LIN {X 0,Y 530.931,Z 527.98,A -85,B 0,C 180,E1 -4418.949,E2 -4418.949} C_VEL
LIN {X 0,Y 531.115,Z 519.525,A -85,B 0,C 180,E1 -4419.907,E2 -4419.907} C_VEL
LIN {X 0,Y 531.409,Z 509.073,A -85,B 0,C 180,E1 -4420.864,E2 -4420.864} C_VEL
LIN {X 0,Y 531.637,Z 497.317,A -85,B 0,C 180,E1 -4421.727,E2 -4421.727} C_VEL
LIN {X 0,Y 531.908,Z 485.378,A -85,B 0,C 180,E1 -4422.4,E2 -4422.4} C_VEL
LIN {X 0,Y 532.176,Z 472.952,A -85,B 0,C 180,E1 -4422.927,E2 -4422.927} C_VEL
LIN {X 0,Y 532.305,Z 460.13,A -85,B 0,C 180,E1 -4423.312,E2 -4423.312} C_VEL
LIN {X 0,Y 530.817,Z 450.091,A -85,B 0,C 180,E1 -4423.545,E2 -4423.545} C_VEL
LIN {X 0,Y 530.994,Z 438.88,A -85,B 0,C 180,E1 -4426.139,E2 -4426.139} C_VEL
LIN {X 0,Y 531.195,Z 426.982,A -85,B 0,C 180,E1 -4428.915,E2 -4428.915} C_VEL
LIN {X 0,Y 531.44,Z 413.99,A -85,B 0,C 180,E1 -4431.982,E2 -4431.982} C_VEL
LIN {X 0,Y 531.748,Z 401.681,A -85,B 0,C 180,E1 -4435.021,E2 -4435.021} C_VEL
LIN {X 0,Y 532.105,Z 389.883,A -85,B 0,C 180,E1 -4438.021,E2 -4438.021} C_VEL
LIN {X 0,Y 532.29,Z 381.917,A -85,B 0,C 180,E1 -4440.115,E2 -4440.115} C_VEL
LIN {X 0,Y 531.009,Z 374.342,A -85,B 0,C 180,E1 -4442.295,E2 -4442.295} C_VEL
LIN {X 0,Y 530.976,Z 374.348,A -85,B 0,C 180,E1 -4444.851,E2 -4444.851} C_VEL
LIN {X 0,Y 530.97,Z 374.344,A -85,B 0,C 180,E1 -4447.508,E2 -4447.508} C_VEL
LIN {X 0,Y 530.953,Z 374.346,A -85,B 0,C 180,E1 -4450.437,E2 -4450.437} C_VEL
LIN {X 0,Y 530.924,Z 374.354,A -85,B 0,C 180,E1 -4453.5,E2 -4453.5} C_VEL
LIN {X 0,Y 530.968,Z 374.344,A -85,B 0,C 180,E1 -4455.624,E2 -4455.624} C_VEL
LIN {X 0,Y 530.968,Z 374.345,A -85,B 0,C 180,E1 -4458.562,E2 -4458.562} C_VEL
LIN {X 0,Y 530.96,Z 374.342,A -85,B 0,C 180,E1 -4461.529,E2 -4461.529} C_VEL
LIN {X 0,Y 530.959,Z 374.35,A -85,B 0,C 180,E1 -4464.38,E2 -4464.38} C_VEL
LIN {X 0,Y 530.972,Z 374.342,A -85,B 0,C 180,E1 -4467.133,E2 -4467.133} C_VEL
LIN {X 0,Y 530.956,Z 374.35,A -85,B 0,C 180,E1 -4469.802,E2 -4469.802} C_VEL
LIN {X 0,Y 530.96,Z 374.344,A -85,B 0,C 180,E1 -4472.48,E2 -4472.48} C_VEL
LIN {X 0,Y 530.949,Z 374.345,A -85,B 0,C 180,E1 -4475.774,E2 -4475.774} C_VEL
LIN {X 0,Y 531.002,Z 374.341,A -85,B 0,C 180,E1 -4479.062,E2 -4479.062} C_VEL
LIN {X 0,Y 530.991,Z 374.34,A -85,B 0,C 180,E1 -4481.479,E2 -4481.479} C_VEL
LIN {X 0,Y 530.999,Z 374.34,A -85,B 0,C 180,E1 -4484.65,E2 -4484.65} C_VEL
LIN {X 0,Y 531.029,Z 374.341,A -85,B 0,C 180,E1 -4487.775,E2 -4487.775} C_VEL
LIN {X 0,Y 530.967,Z 374.344,A -85,B 0,C 180,E1 -4490.091,E2 -4490.091} C_VEL
LIN {X 0,Y 531.015,Z 374.343,A -85,B 0,C 180,E1 -4493.159,E2 -4493.159} C_VEL
LIN {X 0,Y 531.104,Z 374.333,A -85,B 0,C 180,E1 -4494.685,E2 -4494.685} C_VEL
LIN {X 0,Y 530.727,Z 374.457,A -85,B 0,C 180,E1 -4497.058,E2 -4497.058} C_VEL
LIN {X 0,Y 530.921,Z 382.02,A -85,B 0,C 180,E1 -4500,E2 -4500} C_VEL
LIN {X 0,Y 530.728,Z 387.746,A -85,B 0,C 180,E1 -4502.277,E2 -4502.277} C_VEL
LIN {X 0,Y 530.796,Z 395.171,A -85,B 0,C 180,E1 -4505.318,E2 -4505.318} C_VEL
LIN {X 0,Y 530.761,Z 402.54,A -85,B 0,C 180,E1 -4508.375,E2 -4508.375} C_VEL
LIN {X 0,Y 530.722,Z 409.772,A -85,B 0,C 180,E1 -4511.496,E2 -4511.496} C_VEL
LIN {X 0,Y 530.607,Z 417.392,A -85,B 0,C 180,E1 -4514.781,E2 -4514.781} C_VEL
LIN {X 0,Y 530.507,Z 423.618,A -85,B 0,C 180,E1 -4517.537,E2 -4517.537} C_VEL
LIN {X 0,Y 532.297,Z 434.899,A -85,B 0,C 180,E1 -4517.857,E2 -4517.857} C_VEL
LIN {X 0,Y 532.11,Z 445.401,A -85,B 0,C 180,E1 -4518.206,E2 -4518.206} C_VEL
LIN {X 0,Y 531.843,Z 456.316,A -85,B 0,C 180,E1 -4518.69,E2 -4518.69} C_VEL
LIN {X 0,Y 531.666,Z 466.992,A -85,B 0,C 180,E1 -4519.297,E2 -4519.297} C_VEL
LIN {X 0,Y 531.396,Z 479.241,A -85,B 0,C 180,E1 -4520.194,E2 -4520.194} C_VEL
LIN {X 0,Y 531.179,Z 487.4,A -85,B 0,C 180,E1 -4520.93,E2 -4520.93} C_VEL
LIN {X 0,Y 531.018,Z 495.07,A -85,B 0,C 180,E1 -4521.751,E2 -4521.751} C_VEL
LIN {X 0,Y 530.803,Z 503.072,A -85,B 0,C 180,E1 -4522.785,E2 -4522.785} C_VEL
LIN {X 0,Y 530.72,Z 508.892,A -85,B 0,C 180,E1 -4523.683,E2 -4523.683} C_VEL
LIN {X 0,Y 530.572,Z 514.196,A -85,B 0,C 180,E1 -4524.661,E2 -4524.661} C_VEL
LIN {X 0,Y 530.495,Z 519.722,A -85,B 0,C 180,E1 -4525.924,E2 -4525.924} C_VEL
LIN {X 0,Y 530.446,Z 524.375,A -85,B 0,C 180,E1 -4527.414,E2 -4527.414} C_VEL
LIN {X 0,Y 530.399,Z 527.522,A -85,B 0,C 180,E1 -4529.01,E2 -4529.01} C_VEL
LIN {X 0,Y 530.384,Z 528.904,A -85,B 0,C 180,E1 -4530.536,E2 -4530.536} C_VEL
LIN {X 0,Y 530.378,Z 528.658,A -85,B 0,C 180,E1 -4532.008,E2 -4532.008} C_VEL
LIN {X 0,Y 530.368,Z 527.083,A -85,B 0,C 180,E1 -4533.402,E2 -4533.402} C_VEL
LIN {X 0,Y 530.425,Z 524.169,A -85,B 0,C 180,E1 -4534.765,E2 -4534.765} C_VEL
LIN {X 0,Y 530.503,Z 519.993,A -85,B 0,C 180,E1 -4536.087,E2 -4536.087} C_VEL
LIN {X 0,Y 530.589,Z 514.554,A -85,B 0,C 180,E1 -4537.368,E2 -4537.368} C_VEL
LIN {X 0,Y 530.61,Z 512.566,A -85,B 0,C 180,E1 -4537.759,E2 -4537.759} C_VEL
LIN {X 0,Y 529.975,Z 509.631,A -85,B 0,C 180,E1 -4538.31,E2 -4538.31} C_VEL
LIN {X 0,Y 527.214,Z 504.519,A -85,B 0,C 180,E1 -4539.183,E2 -4539.183} C_VEL
LIN {X 0,Y 524.518,Z 498.801,A -85,B 0,C 180,E1 -4540.017,E2 -4540.017} C_VEL
LIN {X 0,Y 523.985,Z 494.917,A -85,B 0,C 180,E1 -4540.501,E2 -4540.501} C_VEL
LIN {X 0,Y 524.222,Z 485.978,A -85,B 0,C 180,E1 -4541.449,E2 -4541.449} C_VEL
LIN {X 0,Y 524.451,Z 476.161,A -85,B 0,C 180,E1 -4542.302,E2 -4542.302} C_VEL
LIN {X 0,Y 524.7,Z 464.968,A -85,B 0,C 180,E1 -4543.087,E2 -4543.087} C_VEL
LIN {X 0,Y 524.982,Z 453.047,A -85,B 0,C 180,E1 -4543.735,E2 -4543.735} C_VEL
LIN {X 0,Y 525.289,Z 439.587,A -85,B 0,C 180,E1 -4544.272,E2 -4544.272} C_VEL
LIN {X 0,Y 525.146,Z 433.464,A -85,B 0,C 180,E1 -4544.464,E2 -4544.464} C_VEL
LIN {X 0,Y 523.424,Z 423.693,A -85,B 0,C 180,E1 -4544.738,E2 -4544.738} C_VEL
LIN {X 0,Y 523.487,Z 417.312,A -85,B 0,C 180,E1 -4547.594,E2 -4547.594} C_VEL
LIN {X 0,Y 523.565,Z 410.89,A -85,B 0,C 180,E1 -4550.403,E2 -4550.403} C_VEL
LIN {X 0,Y 523.64,Z 403.479,A -85,B 0,C 180,E1 -4553.637,E2 -4553.637} C_VEL
LIN {X 0,Y 523.705,Z 396.674,A -85,B 0,C 180,E1 -4556.617,E2 -4556.617} C_VEL
LIN {X 0,Y 523.769,Z 390.415,A -85,B 0,C 180,E1 -4559.342,E2 -4559.342} C_VEL
LIN {X 0,Y 523.781,Z 383.555,A -85,B 0,C 180,E1 -4562.322,E2 -4562.322} C_VEL
LIN {X 0,Y 523.889,Z 376.361,A -85,B 0,C 180,E1 -4565.425,E2 -4565.425} C_VEL
LIN {X 0,Y 523.971,Z 375.22,A -85,B 0,C 180,E1 -4565.962,E2 -4565.962} C_VEL
LIN {X 0,Y 523.948,Z 375.223,A -85,B 0,C 180,E1 -4568.765,E2 -4568.765} C_VEL
LIN {X 0,Y 523.937,Z 375.22,A -85,B 0,C 180,E1 -4571.219,E2 -4571.219} C_VEL
LIN {X 0,Y 523.93,Z 375.226,A -85,B 0,C 180,E1 -4573.637,E2 -4573.637} C_VEL
LIN {X 0,Y 523.941,Z 375.219,A -85,B 0,C 180,E1 -4576.027,E2 -4576.027} C_VEL
LIN {X 0,Y 524.014,Z 375.215,A -85,B 0,C 180,E1 -4578.393,E2 -4578.393} C_VEL
LIN {X 0,Y 524.001,Z 375.217,A -85,B 0,C 180,E1 -4581.514,E2 -4581.514} C_VEL
LIN {X 0,Y 524.073,Z 375.209,A -85,B 0,C 180,E1 -4584.612,E2 -4584.612} C_VEL
LIN {X 0,Y 524.106,Z 375.204,A -85,B 0,C 180,E1 -4587.693,E2 -4587.693} C_VEL
LIN {X 0,Y 524.117,Z 375.253,A -85,B 0,C 180,E1 -4590.286,E2 -4590.286} C_VEL
LIN {X 0,Y 524.079,Z 379.167,A -85,B 0,C 180,E1 -4592.304,E2 -4592.304} C_VEL
LIN {X 0,Y 523.878,Z 385.251,A -85,B 0,C 180,E1 -4595.387,E2 -4595.387} C_VEL
LIN {X 0,Y 523.809,Z 389.903,A -85,B 0,C 180,E1 -4597.709,E2 -4597.709} C_VEL
LIN {X 0,Y 523.734,Z 396.172,A -85,B 0,C 180,E1 -4600.826,E2 -4600.826} C_VEL
LIN {X 0,Y 523.615,Z 402.623,A -85,B 0,C 180,E1 -4603.979,E2 -4603.979} C_VEL
LIN {X 0,Y 523.496,Z 409.248,A -85,B 0,C 180,E1 -4607.176,E2 -4607.176} C_VEL
LIN {X 0,Y 523.382,Z 416.011,A -85,B 0,C 180,E1 -4610.432,E2 -4610.432} C_VEL
LIN {X 0,Y 523.417,Z 419.782,A -85,B 0,C 180,E1 -4612.22,E2 -4612.22} C_VEL
LIN {X 0,Y 524.68,Z 430.393,A -85,B 0,C 180,E1 -4612.57,E2 -4612.57} C_VEL
LIN {X 0,Y 524.396,Z 441.937,A -85,B 0,C 180,E1 -4613.077,E2 -4613.077} C_VEL
LIN {X 0,Y 524.2,Z 450.946,A -85,B 0,C 180,E1 -4613.609,E2 -4613.609} C_VEL
LIN {X 0,Y 524.051,Z 459.242,A -85,B 0,C 180,E1 -4614.226,E2 -4614.226} C_VEL
LIN {X 0,Y 523.927,Z 466.514,A -85,B 0,C 180,E1 -4614.887,E2 -4614.887} C_VEL
LIN {X 0,Y 523.77,Z 472.963,A -85,B 0,C 180,E1 -4615.591,E2 -4615.591} C_VEL
LIN {X 0,Y 523.648,Z 479.751,A -85,B 0,C 180,E1 -4616.501,E2 -4616.501} C_VEL
LIN {X 0,Y 523.529,Z 485.076,A -85,B 0,C 180,E1 -4617.38,E2 -4617.38} C_VEL
LIN {X 0,Y 523.502,Z 488.386,A -85,B 0,C 180,E1 -4618.023,E2 -4618.023} C_VEL
LIN {X 0,Y 523.448,Z 493.123,A -85,B 0,C 180,E1 -4619.225,E2 -4619.225} C_VEL
LIN {X 0,Y 523.384,Z 496.023,A -85,B 0,C 180,E1 -4620.232,E2 -4620.232} C_VEL
LIN {X 0,Y 523.311,Z 497.153,A -85,B 0,C 180,E1 -4620.739,E2 -4620.739} C_VEL
LIN {X 0,Y 523.263,Z 499.086,A -85,B 0,C 180,E1 -4622.204,E2 -4622.204} C_VEL
LIN {X 0,Y 523.294,Z 499.2,A -85,B 0,C 180,E1 -4623.626,E2 -4623.626} C_VEL
LIN {X 0,Y 523.291,Z 498.686,A -85,B 0,C 180,E1 -4624.335,E2 -4624.335} C_VEL
LIN {X 0,Y 523.311,Z 497.339,A -85,B 0,C 180,E1 -4625.271,E2 -4625.271} C_VEL
LIN {X 0,Y 523.396,Z 494.851,A -85,B 0,C 180,E1 -4626.326,E2 -4626.326} C_VEL
LIN {X 0,Y 523.438,Z 492.137,A -85,B 0,C 180,E1 -4627.168,E2 -4627.168} C_VEL
LIN {X 0,Y 523.506,Z 488.098,A -85,B 0,C 180,E1 -4628.134,E2 -4628.134} C_VEL
LIN {X 0,Y 523.605,Z 482.896,A -85,B 0,C 180,E1 -4629.109,E2 -4629.109} C_VEL
LIN {X 0,Y 523.755,Z 476.136,A -85,B 0,C 180,E1 -4630.106,E2 -4630.106} C_VEL
LIN {X 0,Y 523.862,Z 468.849,A -85,B 0,C 180,E1 -4630.969,E2 -4630.969} C_VEL
LIN {X 0,Y 524.025,Z 461.627,A -85,B 0,C 180,E1 -4631.668,E2 -4631.668} C_VEL
LIN {X 0,Y 524.242,Z 453.662,A -85,B 0,C 180,E1 -4632.298,E2 -4632.298} C_VEL
LIN {X 0,Y 524.421,Z 445.007,A -85,B 0,C 180,E1 -4632.849,E2 -4632.849} C_VEL
LIN {X 0,Y 524.56,Z 436.043,A -85,B 0,C 180,E1 -4633.296,E2 -4633.296} C_VEL
LIN {X 0,Y 524.48,Z 427.33,A -85,B 0,C 180,E1 -4633.631,E2 -4633.631} C_VEL
LIN {X 0,Y 523.402,Z 419.767,A -85,B 0,C 180,E1 -4633.89,E2 -4633.89} C_VEL
LIN {X 0,Y 523.452,Z 413.7,A -85,B 0,C 180,E1 -4636.785,E2 -4636.785} C_VEL
LIN {X 0,Y 523.488,Z 408.426,A -85,B 0,C 180,E1 -4639.374,E2 -4639.374} C_VEL
LIN {X 0,Y 523.587,Z 402.331,A -85,B 0,C 180,E1 -4642.363,E2 -4642.363} C_VEL
LIN {X 0,Y 523.658,Z 397.039,A -85,B 0,C 180,E1 -4644.948,E2 -4644.948} C_VEL
LIN {X 0,Y 523.73,Z 391.464,A -85,B 0,C 180,E1 -4647.71,E2 -4647.71} C_VEL
LIN {X 0,Y 523.83,Z 385.498,A -85,B 0,C 180,E1 -4650.695,E2 -4650.695} C_VEL
LIN {X 0,Y 523.929,Z 381.209,A -85,B 0,C 180,E1 -4652.866,E2 -4652.866} C_VEL
LIN {X 0,Y 524.023,Z 375.454,A -85,B 0,C 180,E1 -4655.774,E2 -4655.774} C_VEL
LIN {X 0,Y 523.965,Z 375.222,A -85,B 0,C 180,E1 -4656.272,E2 -4656.272} C_VEL
LIN {X 0,Y 523.936,Z 375.223,A -85,B 0,C 180,E1 -4658.767,E2 -4658.767} C_VEL
LIN {X 0,Y 523.933,Z 375.224,A -85,B 0,C 180,E1 -4661.22,E2 -4661.22} C_VEL
LIN {X 0,Y 523.918,Z 375.226,A -85,B 0,C 180,E1 -4663.639,E2 -4663.639} C_VEL
LIN {X 0,Y 523.929,Z 375.226,A -85,B 0,C 180,E1 -4666.028,E2 -4666.028} C_VEL
LIN {X 0,Y 523.995,Z 375.216,A -85,B 0,C 180,E1 -4668.394,E2 -4668.394} C_VEL
LIN {X 0,Y 523.986,Z 375.217,A -85,B 0,C 180,E1 -4671.516,E2 -4671.516} C_VEL
LIN {X 0,Y 524.083,Z 375.203,A -85,B 0,C 180,E1 -4674.614,E2 -4674.614} C_VEL
LIN {X 0,Y 524.095,Z 375.203,A -85,B 0,C 180,E1 -4677.695,E2 -4677.695} C_VEL
LIN {X 0,Y 524.106,Z 375.202,A -85,B 0,C 180,E1 -4680.769,E2 -4680.769} C_VEL
LIN {X 0,Y 524.056,Z 375.208,A -85,B 0,C 180,E1 -4683.075,E2 -4683.075} C_VEL
LIN {X 0,Y 524.032,Z 375.21,A -85,B 0,C 180,E1 -4686.159,E2 -4686.159} C_VEL
LIN {X 0,Y 523.988,Z 375.214,A -85,B 0,C 180,E1 -4689.262,E2 -4689.262} C_VEL
LIN {X 0,Y 524.019,Z 375.211,A -85,B 0,C 180,E1 -4691.763,E2 -4691.763} C_VEL
LIN {X 0,Y 523.97,Z 375.218,A -85,B 0,C 180,E1 -4695.054,E2 -4695.054} C_VEL
LIN {X 0,Y 523.948,Z 375.223,A -85,B 0,C 180,E1 -4697.97,E2 -4697.97} C_VEL
LIN {X 0,Y 523.951,Z 375.221,A -85,B 0,C 180,E1 -4700.411,E2 -4700.411} C_VEL
LIN {X 0,Y 523.929,Z 375.223,A -85,B 0,C 180,E1 -4702.893,E2 -4702.893} C_VEL
LIN {X 0,Y 523.965,Z 375.221,A -85,B 0,C 180,E1 -4706.022,E2 -4706.022} C_VEL
LIN {X 0,Y 523.931,Z 375.223,A -85,B 0,C 180,E1 -4708.875,E2 -4708.875} C_VEL
LIN {X 0,Y 523.913,Z 375.225,A -85,B 0,C 180,E1 -4711.545,E2 -4711.545} C_VEL
LIN {X 0,Y 523.928,Z 375.224,A -85,B 0,C 180,E1 -4714.291,E2 -4714.291} C_VEL
LIN {X 0,Y 523.894,Z 375.227,A -85,B 0,C 180,E1 -4717.134,E2 -4717.134} C_VEL
LIN {X 0,Y 523.952,Z 375.22,A -85,B 0,C 180,E1 -4720.136,E2 -4720.136} C_VEL
LIN {X 0,Y 523.912,Z 375.227,A -85,B 0,C 180,E1 -4723.168,E2 -4723.168} C_VEL
LIN {X 0,Y 523.927,Z 375.223,A -85,B 0,C 180,E1 -4725.774,E2 -4725.774} C_VEL
LIN {X 0,Y 523.949,Z 375.223,A -85,B 0,C 180,E1 -4728.912,E2 -4728.912} C_VEL
LIN {X 0,Y 523.906,Z 375.226,A -85,B 0,C 180,E1 -4731.901,E2 -4731.901} C_VEL
LIN {X 0,Y 523.93,Z 375.224,A -85,B 0,C 180,E1 -4734.911,E2 -4734.911} C_VEL
LIN {X 0,Y 523.975,Z 375.332,A -85,B 0,C 180,E1 -4737.442,E2 -4737.442} C_VEL
LIN {X 0,Y 525.212,Z 382.036,A -85,B 0,C 180,E1 -4739.44,E2 -4739.44} C_VEL
LIN {X 0,Y 525.262,Z 386.946,A -85,B 0,C 180,E1 -4740.805,E2 -4740.805} C_VEL
LIN {X 0,Y 524.915,Z 396.536,A -85,B 0,C 180,E1 -4743.353,E2 -4743.353} C_VEL
LIN {X 0,Y 524.574,Z 408.028,A -85,B 0,C 180,E1 -4746.304,E2 -4746.304} C_VEL
LIN {X 0,Y 524.243,Z 419.584,A -85,B 0,C 180,E1 -4749.193,E2 -4749.193} C_VEL
LIN {X 0,Y 524.036,Z 432.384,A -85,B 0,C 180,E1 -4752.214,E2 -4752.214} C_VEL
LIN {X 0,Y 523.855,Z 445.336,A -85,B 0,C 180,E1 -4755.234,E2 -4755.234} C_VEL
LIN {X 0,Y 523.765,Z 449.924,A -85,B 0,C 180,E1 -4756.298,E2 -4756.298} C_VEL
LIN {X 0,Y 525.384,Z 461.083,A -85,B 0,C 180,E1 -4756.562,E2 -4756.562} C_VEL
LIN {X 0,Y 525.185,Z 473.533,A -85,B 0,C 180,E1 -4756.951,E2 -4756.951} C_VEL
LIN {X 0,Y 524.916,Z 484.759,A -85,B 0,C 180,E1 -4757.436,E2 -4757.436} C_VEL
LIN {X 0,Y 524.636,Z 496.338,A -85,B 0,C 180,E1 -4758.087,E2 -4758.087} C_VEL
LIN {X 0,Y 524.442,Z 507.516,A -85,B 0,C 180,E1 -4758.895,E2 -4758.895} C_VEL
LIN {X 0,Y 524.157,Z 517.303,A -85,B 0,C 180,E1 -4759.769,E2 -4759.769} C_VEL
LIN {X 0,Y 523.928,Z 526.218,A -85,B 0,C 180,E1 -4760.739,E2 -4760.739} C_VEL
LIN {X 0,Y 523.722,Z 534.907,A -85,B 0,C 180,E1 -4761.902,E2 -4761.902} C_VEL
LIN {X 0,Y 523.573,Z 541.849,A -85,B 0,C 180,E1 -4763.063,E2 -4763.063} C_VEL
LIN {X 0,Y 523.543,Z 547.372,A -85,B 0,C 180,E1 -4764.224,E2 -4764.224} C_VEL
LIN {X 0,Y 523.36,Z 551.682,A -85,B 0,C 180,E1 -4765.38,E2 -4765.38} C_VEL
LIN {X 0,Y 523.443,Z 553.965,A -85,B 0,C 180,E1 -4766.153,E2 -4766.153} C_VEL
LIN {X 0,Y 523.367,Z 555.814,A -85,B 0,C 180,E1 -4766.923,E2 -4766.923} C_VEL
LIN {X 0,Y 523.335,Z 557.198,A -85,B 0,C 180,E1 -4767.693,E2 -4767.693} C_VEL
LIN {X 0,Y 523.25,Z 558.787,A -85,B 0,C 180,E1 -4769.232,E2 -4769.232} C_VEL
LIN {X 0,Y 523.246,Z 559,A -85,B 0,C 180,E1 -4770.002,E2 -4770.002} C_VEL
LIN {X 0,Y 523.275,Z 558.18,A -85,B 0,C 180,E1 -4771.541,E2 -4771.541} C_VEL
LIN {X 0,Y 523.335,Z 557.19,A -85,B 0,C 180,E1 -4772.311,E2 -4772.311} C_VEL
LIN {X 0,Y 523.368,Z 555.803,A -85,B 0,C 180,E1 -4773.081,E2 -4773.081} C_VEL
LIN {X 0,Y 523.442,Z 552.889,A -85,B 0,C 180,E1 -4774.237,E2 -4774.237} C_VEL
LIN {X 0,Y 523.465,Z 548.944,A -85,B 0,C 180,E1 -4775.394,E2 -4775.394} C_VEL
LIN {X 0,Y 523.525,Z 543.706,A -85,B 0,C 180,E1 -4776.582,E2 -4776.582} C_VEL
LIN {X 0,Y 523.667,Z 537.376,A -85,B 0,C 180,E1 -4777.714,E2 -4777.714} C_VEL
LIN {X 0,Y 523.846,Z 529.297,A -85,B 0,C 180,E1 -4778.877,E2 -4778.877} C_VEL
LIN {X 0,Y 524.057,Z 521.061,A -85,B 0,C 180,E1 -4779.847,E2 -4779.847} C_VEL
LIN {X 0,Y 524.316,Z 511.016,A -85,B 0,C 180,E1 -4780.818,E2 -4780.818} C_VEL
LIN {X 0,Y 524.632,Z 499.723,A -85,B 0,C 180,E1 -4781.686,E2 -4781.686} C_VEL
LIN {X 0,Y 524.831,Z 488.494,A -85,B 0,C 180,E1 -4782.373,E2 -4782.373} C_VEL
LIN {X 0,Y 525.135,Z 476.104,A -85,B 0,C 180,E1 -4782.955,E2 -4782.955} C_VEL
LIN {X 0,Y 525.363,Z 462.889,A -85,B 0,C 180,E1 -4783.392,E2 -4783.392} C_VEL
LIN {X 0,Y 524.977,Z 457.876,A -85,B 0,C 180,E1 -4783.526,E2 -4783.526} C_VEL
LIN {X 0,Y 523.756,Z 449.781,A -85,B 0,C 180,E1 -4783.731,E2 -4783.731} C_VEL
LIN {X 0,Y 523.945,Z 438.566,A -85,B 0,C 180,E1 -4786.362,E2 -4786.362} C_VEL
LIN {X 0,Y 524.147,Z 426.663,A -85,B 0,C 180,E1 -4789.179,E2 -4789.179} C_VEL
LIN {X 0,Y 524.441,Z 414.908,A -85,B 0,C 180,E1 -4792.04,E2 -4792.04} C_VEL
LIN {X 0,Y 524.766,Z 403.24,A -85,B 0,C 180,E1 -4794.954,E2 -4794.954} C_VEL
LIN {X 0,Y 525.183,Z 390.057,A -85,B 0,C 180,E1 -4798.364,E2 -4798.364} C_VEL
LIN {X 0,Y 525.367,Z 383.542,A -85,B 0,C 180,E1 -4800.11,E2 -4800.11} C_VEL
LIN {X 0,Y 523.958,Z 375.222,A -85,B 0,C 180,E1 -4802.534,E2 -4802.534} C_VEL
LIN {X 0,Y 523.925,Z 375.223,A -85,B 0,C 180,E1 -4805.227,E2 -4805.227} C_VEL
LIN {X 0,Y 523.919,Z 375.227,A -85,B 0,C 180,E1 -4808.103,E2 -4808.103} C_VEL
LIN {X 0,Y 523.92,Z 375.222,A -85,B 0,C 180,E1 -4811.305,E2 -4811.305} C_VEL
LIN {X 0,Y 523.936,Z 375.219,A -85,B 0,C 180,E1 -4814.689,E2 -4814.689} C_VEL
LIN {X 0,Y 523.913,Z 375.221,A -85,B 0,C 180,E1 -4817.877,E2 -4817.877} C_VEL
LIN {X 0,Y 523.921,Z 375.222,A -85,B 0,C 180,E1 -4821.081,E2 -4821.081} C_VEL
LIN {X 0,Y 523.906,Z 375.223,A -85,B 0,C 180,E1 -4823.825,E2 -4823.825} C_VEL
LIN {X 0,Y 523.918,Z 375.222,A -85,B 0,C 180,E1 -4826.634,E2 -4826.634} C_VEL
LIN {X 0,Y 523.949,Z 375.219,A -85,B 0,C 180,E1 -4829.355,E2 -4829.355} C_VEL
LIN {X 0,Y 523.917,Z 375.221,A -85,B 0,C 180,E1 -4832.295,E2 -4832.295} C_VEL
LIN {X 0,Y 523.897,Z 375.226,A -85,B 0,C 180,E1 -4835.426,E2 -4835.426} C_VEL
LIN {X 0,Y 523.942,Z 375.218,A -85,B 0,C 180,E1 -4837.939,E2 -4837.939} C_VEL
LIN {X 0,Y 523.978,Z 375.22,A -85,B 0,C 180,E1 -4840.408,E2 -4840.408} C_VEL
LIN {X 0,Y 523.971,Z 375.216,A -85,B 0,C 180,E1 -4842.837,E2 -4842.837} C_VEL
LIN {X 0,Y 523.981,Z 375.215,A -85,B 0,C 180,E1 -4845.236,E2 -4845.236} C_VEL
LIN {X 0,Y 524.017,Z 375.209,A -85,B 0,C 180,E1 -4848.394,E2 -4848.394} C_VEL
LIN {X 0,Y 523.948,Z 375.222,A -85,B 0,C 180,E1 -4851.515,E2 -4851.515} C_VEL
LIN {X 0,Y 524.048,Z 375.211,A -85,B 0,C 180,E1 -4854.613,E2 -4854.613} C_VEL
LIN {X 0,Y 523.669,Z 375.428,A -85,B 0,C 180,E1 -4857.115,E2 -4857.115} C_VEL
LIN {X 0,Y 523.879,Z 382.806,A -85,B 0,C 180,E1 -4860,E2 -4860} C_VEL
LIN {X 0,Y 523.662,Z 388.565,A -85,B 0,C 180,E1 -4862.307,E2 -4862.307} C_VEL
LIN {X 0,Y 523.744,Z 394.199,A -85,B 0,C 180,E1 -4864.618,E2 -4864.618} C_VEL
LIN {X 0,Y 523.679,Z 401.576,A -85,B 0,C 180,E1 -4867.712,E2 -4867.712} C_VEL
LIN {X 0,Y 523.619,Z 407.094,A -85,B 0,C 180,E1 -4870.048,E2 -4870.048} C_VEL
LIN {X 0,Y 523.572,Z 412.511,A -85,B 0,C 180,E1 -4872.402,E2 -4872.402} C_VEL
LIN {X 0,Y 523.522,Z 418.186,A -85,B 0,C 180,E1 -4874.858,E2 -4874.858} C_VEL
LIN {X 0,Y 523.445,Z 423.749,A -85,B 0,C 180,E1 -4877.352,E2 -4877.352} C_VEL
LIN {X 0,Y 525.37,Z 435.711,A -85,B 0,C 180,E1 -4877.699,E2 -4877.699} C_VEL
LIN {X 0,Y 525.152,Z 448.719,A -85,B 0,C 180,E1 -4878.161,E2 -4878.161} C_VEL
LIN {X 0,Y 524.83,Z 460.623,A -85,B 0,C 180,E1 -4878.746,E2 -4878.746} C_VEL
LIN {X 0,Y 524.598,Z 471.88,A -85,B 0,C 180,E1 -4879.466,E2 -4879.466} C_VEL
LIN {X 0,Y 524.355,Z 481.646,A -85,B 0,C 180,E1 -4880.244,E2 -4880.244} C_VEL
LIN {X 0,Y 524.113,Z 489.742,A -85,B 0,C 180,E1 -4881.02,E2 -4881.02} C_VEL
LIN {X 0,Y 523.901,Z 497.087,A -85,B 0,C 180,E1 -4881.855,E2 -4881.855} C_VEL
LIN {X 0,Y 523.736,Z 504.746,A -85,B 0,C 180,E1 -4882.901,E2 -4882.901} C_VEL
LIN {X 0,Y 523.592,Z 510.906,A -85,B 0,C 180,E1 -4883.922,E2 -4883.922} C_VEL
LIN {X 0,Y 523.44,Z 516.33,A -85,B 0,C 180,E1 -4885.02,E2 -4885.02} C_VEL
LIN {X 0,Y 523.409,Z 521.329,A -85,B 0,C 180,E1 -4886.302,E2 -4886.302} C_VEL
LIN {X 0,Y 523.335,Z 524.976,A -85,B 0,C 180,E1 -4887.583,E2 -4887.583} C_VEL
LIN {X 0,Y 523.305,Z 527.778,A -85,B 0,C 180,E1 -4889.196,E2 -4889.196} C_VEL
LIN {X 0,Y 523.315,Z 528.473,A -85,B 0,C 180,E1 -4889.795,E2 -4889.795} C_VEL
LIN {X 0,Y 523.281,Z 528.947,A -85,B 0,C 180,E1 -4890.732,E2 -4890.732} C_VEL
LIN {X 0,Y 523.272,Z 528.55,A -85,B 0,C 180,E1 -4892.204,E2 -4892.204} C_VEL
LIN {X 0,Y 523.292,Z 526.766,A -85,B 0,C 180,E1 -4893.624,E2 -4893.624} C_VEL
LIN {X 0,Y 523.329,Z 523.715,A -85,B 0,C 180,E1 -4894.995,E2 -4894.995} C_VEL
LIN {X 0,Y 523.426,Z 519.412,A -85,B 0,C 180,E1 -4896.329,E2 -4896.329} C_VEL
LIN {X 0,Y 523.532,Z 513.794,A -85,B 0,C 180,E1 -4897.624,E2 -4897.624} C_VEL
LIN {X 0,Y 523.638,Z 506.783,A -85,B 0,C 180,E1 -4898.881,E2 -4898.881} C_VEL
LIN {X 0,Y 523.864,Z 498.325,A -85,B 0,C 180,E1 -4900.087,E2 -4900.087} C_VEL
LIN {X 0,Y 523.985,Z 494.917,A -85,B 0,C 180,E1 -4900.501,E2 -4900.501} C_VEL
LIN {X 0,Y 523.445,Z 490.873,A -85,B 0,C 180,E1 -4900.968,E2 -4900.968} C_VEL
LIN {X 0,Y 520.748,Z 484.101,A -85,B 0,C 180,E1 -4901.71,E2 -4901.71} C_VEL
LIN {X 0,Y 518.081,Z 476.865,A -85,B 0,C 180,E1 -4902.398,E2 -4902.398} C_VEL
LIN {X 0,Y 517.579,Z 472.072,A -85,B 0,C 180,E1 -4902.775,E2 -4902.775} C_VEL
LIN {X 0,Y 517.872,Z 460.337,A -85,B 0,C 180,E1 -4903.531,E2 -4903.531} C_VEL
LIN {X 0,Y 518.181,Z 448.806,A -85,B 0,C 180,E1 -4904.103,E2 -4904.103} C_VEL
LIN {X 0,Y 518.424,Z 435.768,A -85,B 0,C 180,E1 -4904.573,E2 -4904.573} C_VEL
LIN {X 0,Y 516.35,Z 423.831,A -85,B 0,C 180,E1 -4904.928,E2 -4904.928} C_VEL
LIN {X 0,Y 516.415,Z 418.568,A -85,B 0,C 180,E1 -4907.298,E2 -4907.298} C_VEL
LIN {X 0,Y 516.501,Z 411.881,A -85,B 0,C 180,E1 -4910.242,E2 -4910.242} C_VEL
LIN {X 0,Y 516.558,Z 404.748,A -85,B 0,C 180,E1 -4913.39,E2 -4913.39} C_VEL
LIN {X 0,Y 516.655,Z 398.582,A -85,B 0,C 180,E1 -4916.101,E2 -4916.101} C_VEL
LIN {X 0,Y 516.71,Z 392.061,A -85,B 0,C 180,E1 -4918.969,E2 -4918.969} C_VEL
LIN {X 0,Y 516.738,Z 384.873,A -85,B 0,C 180,E1 -4922.134,E2 -4922.134} C_VEL
LIN {X 0,Y 516.805,Z 378.075,A -85,B 0,C 180,E1 -4925.065,E2 -4925.065} C_VEL
LIN {X 0,Y 516.902,Z 376.101,A -85,B 0,C 180,E1 -4925.926,E2 -4925.926} C_VEL
LIN {X 0,Y 516.888,Z 376.099,A -85,B 0,C 180,E1 -4928.461,E2 -4928.461} C_VEL
LIN {X 0,Y 516.892,Z 376.098,A -85,B 0,C 180,E1 -4930.953,E2 -4930.953} C_VEL
LIN {X 0,Y 516.905,Z 376.099,A -85,B 0,C 180,E1 -4933.409,E2 -4933.409} C_VEL
LIN {X 0,Y 516.896,Z 376.097,A -85,B 0,C 180,E1 -4935.832,E2 -4935.832} C_VEL
LIN {X 0,Y 516.95,Z 376.09,A -85,B 0,C 180,E1 -4939.026,E2 -4939.026} C_VEL
LIN {X 0,Y 516.979,Z 376.087,A -85,B 0,C 180,E1 -4942.185,E2 -4942.185} C_VEL
LIN {X 0,Y 517.02,Z 376.087,A -85,B 0,C 180,E1 -4944.538,E2 -4944.538} C_VEL
LIN {X 0,Y 517.075,Z 376.079,A -85,B 0,C 180,E1 -4947.661,E2 -4947.661} C_VEL
LIN {X 0,Y 517.089,Z 376.227,A -85,B 0,C 180,E1 -4950.29,E2 -4950.29} C_VEL
LIN {X 0,Y 517.044,Z 380.165,A -85,B 0,C 180,E1 -4952.335,E2 -4952.335} C_VEL
LIN {X 0,Y 516.834,Z 386.28,A -85,B 0,C 180,E1 -4955.46,E2 -4955.46} C_VEL
LIN {X 0,Y 516.752,Z 390.94,A -85,B 0,C 180,E1 -4957.815,E2 -4957.815} C_VEL
LIN {X 0,Y 516.672,Z 397.259,A -85,B 0,C 180,E1 -4960.976,E2 -4960.976} C_VEL
LIN {X 0,Y 516.543,Z 403.706,A -85,B 0,C 180,E1 -4964.174,E2 -4964.174} C_VEL
LIN {X 0,Y 516.416,Z 410.386,A -85,B 0,C 180,E1 -4967.419,E2 -4967.419} C_VEL
LIN {X 0,Y 516.311,Z 417.245,A -85,B 0,C 180,E1 -4970.724,E2 -4970.724} C_VEL
LIN {X 0,Y 516.354,Z 420.001,A -85,B 0,C 180,E1 -4972.049,E2 -4972.049} C_VEL
LIN {X 0,Y 517.737,Z 430.351,A -85,B 0,C 180,E1 -4972.401,E2 -4972.401} C_VEL
LIN {X 0,Y 517.492,Z 441.255,A -85,B 0,C 180,E1 -4972.874,E2 -4972.874} C_VEL
LIN {X 0,Y 517.25,Z 450.502,A -85,B 0,C 180,E1 -4973.415,E2 -4973.415} C_VEL
LIN {X 0,Y 517.076,Z 459.202,A -85,B 0,C 180,E1 -4974.061,E2 -4974.061} C_VEL
LIN {X 0,Y 516.937,Z 466.896,A -85,B 0,C 180,E1 -4974.768,E2 -4974.768} C_VEL
LIN {X 0,Y 516.727,Z 474.126,A -85,B 0,C 180,E1 -4975.581,E2 -4975.581} C_VEL
LIN {X 0,Y 516.586,Z 480.875,A -85,B 0,C 180,E1 -4976.52,E2 -4976.52} C_VEL
LIN {X 0,Y 516.42,Z 486.841,A -85,B 0,C 180,E1 -4977.559,E2 -4977.559} C_VEL
LIN {X 0,Y 516.367,Z 490.849,A -85,B 0,C 180,E1 -4978.446,E2 -4978.446} C_VEL
LIN {X 0,Y 516.362,Z 494.298,A -85,B 0,C 180,E1 -4979.416,E2 -4979.416} C_VEL
LIN {X 0,Y 516.313,Z 496.533,A -85,B 0,C 180,E1 -4980.238,E2 -4980.238} C_VEL
LIN {X 0,Y 516.197,Z 498.334,A -85,B 0,C 180,E1 -4981.153,E2 -4981.153} C_VEL
LIN {X 0,Y 516.199,Z 499.6,A -85,B 0,C 180,E1 -4982.422,E2 -4982.422} C_VEL
LIN {X 0,Y 516.189,Z 499.812,A -85,B 0,C 180,E1 -4982.995,E2 -4982.995} C_VEL
LIN {X 0,Y 516.212,Z 499.483,A -85,B 0,C 180,E1 -4983.928,E2 -4983.928} C_VEL
LIN {X 0,Y 516.239,Z 497.878,A -85,B 0,C 180,E1 -4985.232,E2 -4985.232} C_VEL
LIN {X 0,Y 516.344,Z 494.629,A -85,B 0,C 180,E1 -4986.578,E2 -4986.578} C_VEL
LIN {X 0,Y 516.385,Z 492.378,A -85,B 0,C 180,E1 -4987.272,E2 -4987.272} C_VEL
LIN {X 0,Y 516.492,Z 486.985,A -85,B 0,C 180,E1 -4988.512,E2 -4988.512} C_VEL
LIN {X 0,Y 516.602,Z 480.999,A -85,B 0,C 180,E1 -4989.561,E2 -4989.561} C_VEL
LIN {X 0,Y 516.769,Z 473.995,A -85,B 0,C 180,E1 -4990.535,E2 -4990.535} C_VEL
LIN {X 0,Y 516.942,Z 465.914,A -85,B 0,C 180,E1 -4991.433,E2 -4991.433} C_VEL
LIN {X 0,Y 517.202,Z 456.374,A -85,B 0,C 180,E1 -4992.267,E2 -4992.267} C_VEL
LIN {X 0,Y 517.44,Z 445.973,A -85,B 0,C 180,E1 -4992.963,E2 -4992.963} C_VEL
LIN {X 0,Y 517.622,Z 435.978,A -85,B 0,C 180,E1 -4993.469,E2 -4993.469} C_VEL
LIN {X 0,Y 517.541,Z 427.826,A -85,B 0,C 180,E1 -4993.787,E2 -4993.787} C_VEL
LIN {X 0,Y 516.341,Z 420.016,A -85,B 0,C 180,E1 -4994.063,E2 -4994.063} C_VEL
LIN {X 0,Y 516.387,Z 413.267,A -85,B 0,C 180,E1 -4997.298,E2 -4997.298} C_VEL
LIN {X 0,Y 516.43,Z 407.387,A -85,B 0,C 180,E1 -5000.237,E2 -5000.237} C_VEL
LIN {X 0,Y 516.538,Z 401.298,A -85,B 0,C 180,E1 -5003.226,E2 -5003.226} C_VEL
LIN {X 0,Y 516.63,Z 395.497,A -85,B 0,C 180,E1 -5006.1,E2 -5006.1} C_VEL
LIN {X 0,Y 516.719,Z 389.826,A -85,B 0,C 180,E1 -5008.962,E2 -5008.962} C_VEL
LIN {X 0,Y 516.876,Z 383.649,A -85,B 0,C 180,E1 -5012.099,E2 -5012.099} C_VEL
LIN {X 0,Y 516.971,Z 377.826,A -85,B 0,C 180,E1 -5015.075,E2 -5015.075} C_VEL
LIN {X 0,Y 516.952,Z 376.095,A -85,B 0,C 180,E1 -5016.037,E2 -5016.037} C_VEL
LIN {X 0,Y 516.893,Z 376.103,A -85,B 0,C 180,E1 -5019.298,E2 -5019.298} C_VEL
LIN {X 0,Y 516.907,Z 376.099,A -85,B 0,C 180,E1 -5022.596,E2 -5022.596} C_VEL
LIN {X 0,Y 516.926,Z 376.096,A -85,B 0,C 180,E1 -5025.03,E2 -5025.03} C_VEL
LIN {X 0,Y 516.978,Z 376.089,A -85,B 0,C 180,E1 -5028.234,E2 -5028.234} C_VEL
LIN {X 0,Y 516.95,Z 376.094,A -85,B 0,C 180,E1 -5031.4,E2 -5031.4} C_VEL
LIN {X 0,Y 517.044,Z 376.08,A -85,B 0,C 180,E1 -5034.54,E2 -5034.54} C_VEL
LIN {X 0,Y 517.066,Z 376.079,A -85,B 0,C 180,E1 -5037.663,E2 -5037.663} C_VEL
LIN {X 0,Y 517.075,Z 376.077,A -85,B 0,C 180,E1 -5040.779,E2 -5040.779} C_VEL
LIN {X 0,Y 517.023,Z 376.085,A -85,B 0,C 180,E1 -5043.117,E2 -5043.117} C_VEL
LIN {X 0,Y 516.994,Z 376.086,A -85,B 0,C 180,E1 -5046.244,E2 -5046.244} C_VEL
LIN {X 0,Y 516.943,Z 376.091,A -85,B 0,C 180,E1 -5049.39,E2 -5049.39} C_VEL
LIN {X 0,Y 516.978,Z 376.088,A -85,B 0,C 180,E1 -5051.836,E2 -5051.836} C_VEL
LIN {X 0,Y 516.923,Z 376.097,A -85,B 0,C 180,E1 -5055.149,E2 -5055.149} C_VEL
LIN {X 0,Y 516.908,Z 376.097,A -85,B 0,C 180,E1 -5058.223,E2 -5058.223} C_VEL
LIN {X 0,Y 516.895,Z 376.101,A -85,B 0,C 180,E1 -5060.702,E2 -5060.702} C_VEL
LIN {X 0,Y 516.873,Z 376.104,A -85,B 0,C 180,E1 -5063.224,E2 -5063.224} C_VEL
LIN {X 0,Y 516.924,Z 376.096,A -85,B 0,C 180,E1 -5066.198,E2 -5066.198} C_VEL
LIN {X 0,Y 516.916,Z 376.095,A -85,B 0,C 180,E1 -5069.305,E2 -5069.305} C_VEL
LIN {X 0,Y 516.882,Z 376.101,A -85,B 0,C 180,E1 -5072.546,E2 -5072.546} C_VEL
LIN {X 0,Y 516.866,Z 376.105,A -85,B 0,C 180,E1 -5075.334,E2 -5075.334} C_VEL
LIN {X 0,Y 516.865,Z 376.105,A -85,B 0,C 180,E1 -5077.945,E2 -5077.945} C_VEL
LIN {X 0,Y 516.888,Z 376.103,A -85,B 0,C 180,E1 -5080.742,E2 -5080.742} C_VEL
LIN {X 0,Y 516.869,Z 376.102,A -85,B 0,C 180,E1 -5083.905,E2 -5083.905} C_VEL
LIN {X 0,Y 516.868,Z 376.106,A -85,B 0,C 180,E1 -5086.109,E2 -5086.109} C_VEL
LIN {X 0,Y 516.892,Z 376.1,A -85,B 0,C 180,E1 -5089.263,E2 -5089.263} C_VEL
LIN {X 0,Y 516.871,Z 376.102,A -85,B 0,C 180,E1 -5092.059,E2 -5092.059} C_VEL
LIN {X 0,Y 516.887,Z 376.103,A -85,B 0,C 180,E1 -5095.179,E2 -5095.179} C_VEL
LIN {X 0,Y 516.93,Z 376.196,A -85,B 0,C 180,E1 -5097.173,E2 -5097.173} C_VEL
LIN {X 0,Y 518.29,Z 383.649,A -85,B 0,C 180,E1 -5099.439,E2 -5099.439} C_VEL
LIN {X 0,Y 518.327,Z 388.435,A -85,B 0,C 180,E1 -5100.785,E2 -5100.785} C_VEL
LIN {X 0,Y 517.87,Z 398.845,A -85,B 0,C 180,E1 -5103.597,E2 -5103.597} C_VEL
LIN {X 0,Y 517.505,Z 411.276,A -85,B 0,C 180,E1 -5106.809,E2 -5106.809} C_VEL
LIN {X 0,Y 517.174,Z 422.525,A -85,B 0,C 180,E1 -5109.663,E2 -5109.663} C_VEL
LIN {X 0,Y 516.936,Z 436.542,A -85,B 0,C 180,E1 -5113.006,E2 -5113.006} C_VEL
LIN {X 0,Y 516.7,Z 449.805,A -85,B 0,C 180,E1 -5116.132,E2 -5116.132} C_VEL
LIN {X 0,Y 518.423,Z 461.913,A -85,B 0,C 180,E1 -5116.428,E2 -5116.428} C_VEL
LIN {X 0,Y 518.189,Z 475.35,A -85,B 0,C 180,E1 -5116.871,E2 -5116.871} C_VEL
LIN {X 0,Y 517.915,Z 486.074,A -85,B 0,C 180,E1 -5117.363,E2 -5117.363} C_VEL
LIN {X 0,Y 517.611,Z 496.923,A -85,B 0,C 180,E1 -5118.002,E2 -5118.002} C_VEL
LIN {X 0,Y 517.4,Z 508.165,A -85,B 0,C 180,E1 -5118.841,E2 -5118.841} C_VEL
LIN {X 0,Y 517.045,Z 518.767,A -85,B 0,C 180,E1 -5119.824,E2 -5119.824} C_VEL
LIN {X 0,Y 516.823,Z 527.347,A -85,B 0,C 180,E1 -5120.808,E2 -5120.808} C_VEL
LIN {X 0,Y 516.615,Z 535.7,A -85,B 0,C 180,E1 -5121.986,E2 -5121.986} C_VEL
LIN {X 0,Y 516.505,Z 541.412,A -85,B 0,C 180,E1 -5122.968,E2 -5122.968} C_VEL
LIN {X 0,Y 516.453,Z 546.986,A -85,B 0,C 180,E1 -5124.144,E2 -5124.144} C_VEL
LIN {X 0,Y 516.271,Z 551.35,A -85,B 0,C 180,E1 -5125.317,E2 -5125.317} C_VEL
LIN {X 0,Y 516.354,Z 553.672,A -85,B 0,C 180,E1 -5126.1,E2 -5126.1} C_VEL
LIN {X 0,Y 516.282,Z 555.544,A -85,B 0,C 180,E1 -5126.88,E2 -5126.88} C_VEL
LIN {X 0,Y 516.261,Z 556.949,A -85,B 0,C 180,E1 -5127.661,E2 -5127.661} C_VEL
LIN {X 0,Y 516.16,Z 558.555,A -85,B 0,C 180,E1 -5129.222,E2 -5129.222} C_VEL
LIN {X 0,Y 516.154,Z 558.772,A -85,B 0,C 180,E1 -5130.002,E2 -5130.002} C_VEL
LIN {X 0,Y 516.192,Z 557.943,A -85,B 0,C 180,E1 -5131.562,E2 -5131.562} C_VEL
LIN {X 0,Y 516.262,Z 556.943,A -85,B 0,C 180,E1 -5132.342,E2 -5132.342} C_VEL
LIN {X 0,Y 516.283,Z 555.537,A -85,B 0,C 180,E1 -5133.123,E2 -5133.123} C_VEL
LIN {X 0,Y 516.327,Z 552.586,A -85,B 0,C 180,E1 -5134.295,E2 -5134.295} C_VEL
LIN {X 0,Y 516.406,Z 548.589,A -85,B 0,C 180,E1 -5135.468,E2 -5135.468} C_VEL
LIN {X 0,Y 516.446,Z 543.251,A -85,B 0,C 180,E1 -5136.681,E2 -5136.681} C_VEL
LIN {X 0,Y 516.58,Z 536.941,A -85,B 0,C 180,E1 -5137.821,E2 -5137.821} C_VEL
LIN {X 0,Y 516.808,Z 528.851,A -85,B 0,C 180,E1 -5138.999,E2 -5138.999} C_VEL
LIN {X 0,Y 516.997,Z 520.595,A -85,B 0,C 180,E1 -5139.983,E2 -5139.983} C_VEL
LIN {X 0,Y 517.317,Z 510.524,A -85,B 0,C 180,E1 -5140.966,E2 -5140.966} C_VEL
LIN {X 0,Y 517.579,Z 500.537,A -85,B 0,C 180,E1 -5141.754,E2 -5141.754} C_VEL
LIN {X 0,Y 517.824,Z 489.244,A -85,B 0,C 180,E1 -5142.468,E2 -5142.468} C_VEL
LIN {X 0,Y 518.121,Z 477.704,A -85,B 0,C 180,E1 -5143.034,E2 -5143.034} C_VEL
LIN {X 0,Y 518.402,Z 464.702,A -85,B 0,C 180,E1 -5143.501,E2 -5143.501} C_VEL
LIN {X 0,Y 518.164,Z 459.483,A -85,B 0,C 180,E1 -5143.647,E2 -5143.647} C_VEL
LIN {X 0,Y 516.693,Z 449.576,A -85,B 0,C 180,E1 -5143.897,E2 -5143.897} C_VEL
LIN {X 0,Y 516.894,Z 438.252,A -85,B 0,C 180,E1 -5146.592,E2 -5146.592} C_VEL
LIN {X 0,Y 517.119,Z 426.47,A -85,B 0,C 180,E1 -5149.451,E2 -5149.451} C_VEL
LIN {X 0,Y 517.43,Z 414.767,A -85,B 0,C 180,E1 -5152.354,E2 -5152.354} C_VEL
LIN {X 0,Y 517.794,Z 403.144,A -85,B 0,C 180,E1 -5155.313,E2 -5155.313} C_VEL
LIN {X 0,Y 518.213,Z 391.643,A -85,B 0,C 180,E1 -5158.339,E2 -5158.339} C_VEL
LIN {X 0,Y 518.447,Z 385.159,A -85,B 0,C 180,E1 -5160.105,E2 -5160.105} C_VEL
LIN {X 0,Y 517.411,Z 378.714,A -85,B 0,C 180,E1 -5161.989,E2 -5161.989} C_VEL
LIN {X 0,Y 516.919,Z 376.097,A -85,B 0,C 180,E1 -5162.829,E2 -5162.829} C_VEL
LIN {X 0,Y 516.875,Z 376.101,A -85,B 0,C 180,E1 -5165.781,E2 -5165.781} C_VEL
LIN {X 0,Y 516.883,Z 376.1,A -85,B 0,C 180,E1 -5168.717,E2 -5168.717} C_VEL
LIN {X 0,Y 516.849,Z 376.108,A -85,B 0,C 180,E1 -5171.783,E2 -5171.783} C_VEL
LIN {X 0,Y 516.902,Z 376.098,A -85,B 0,C 180,E1 -5175.007,E2 -5175.007} C_VEL
LIN {X 0,Y 516.893,Z 376.097,A -85,B 0,C 180,E1 -5178.402,E2 -5178.402} C_VEL
LIN {X 0,Y 516.885,Z 376.096,A -85,B 0,C 180,E1 -5181.284,E2 -5181.284} C_VEL
LIN {X 0,Y 516.876,Z 376.104,A -85,B 0,C 180,E1 -5184.22,E2 -5184.22} C_VEL
LIN {X 0,Y 516.886,Z 376.096,A -85,B 0,C 180,E1 -5187.052,E2 -5187.052} C_VEL
LIN {X 0,Y 516.871,Z 376.104,A -85,B 0,C 180,E1 -5189.795,E2 -5189.795} C_VEL
LIN {X 0,Y 516.872,Z 376.099,A -85,B 0,C 180,E1 -5192.464,E2 -5192.464} C_VEL
LIN {X 0,Y 516.859,Z 376.101,A -85,B 0,C 180,E1 -5195.65,E2 -5195.65} C_VEL
LIN {X 0,Y 516.889,Z 376.101,A -85,B 0,C 180,E1 -5198.462,E2 -5198.462} C_VEL
LIN {X 0,Y 516.905,Z 376.096,A -85,B 0,C 180,E1 -5200.955,E2 -5200.955} C_VEL
LIN {X 0,Y 516.917,Z 376.094,A -85,B 0,C 180,E1 -5203.41,E2 -5203.41} C_VEL
LIN {X 0,Y 516.896,Z 376.102,A -85,B 0,C 180,E1 -5205.833,E2 -5205.833} C_VEL
LIN {X 0,Y 516.946,Z 376.093,A -85,B 0,C 180,E1 -5209.027,E2 -5209.027} C_VEL
LIN {X 0,Y 516.924,Z 376.093,A -85,B 0,C 180,E1 -5212.186,E2 -5212.186} C_VEL
LIN {X 0,Y 516.997,Z 376.088,A -85,B 0,C 180,E1 -5214.539,E2 -5214.539} C_VEL
LIN {X 0,Y 516.621,Z 376.195,A -85,B 0,C 180,E1 -5217.076,E2 -5217.076} C_VEL
LIN {X 0,Y 516.839,Z 383.607,A -85,B 0,C 180,E1 -5220,E2 -5220} C_VEL
LIN {X 0,Y 516.599,Z 389.412,A -85,B 0,C 180,E1 -5222.339,E2 -5222.339} C_VEL
LIN {X 0,Y 516.68,Z 395.074,A -85,B 0,C 180,E1 -5224.681,E2 -5224.681} C_VEL
LIN {X 0,Y 516.618,Z 402.434,A -85,B 0,C 180,E1 -5227.818,E2 -5227.818} C_VEL
LIN {X 0,Y 516.576,Z 409.895,A -85,B 0,C 180,E1 -5230.98,E2 -5230.98} C_VEL
LIN {X 0,Y 516.46,Z 417.216,A -85,B 0,C 180,E1 -5234.178,E2 -5234.178} C_VEL
LIN {X 0,Y 516.371,Z 423.979,A -85,B 0,C 180,E1 -5237.168,E2 -5237.168} C_VEL
LIN {X 0,Y 518.467,Z 436.608,A -85,B 0,C 180,E1 -5237.543,E2 -5237.543} C_VEL
LIN {X 0,Y 518.219,Z 449.052,A -85,B 0,C 180,E1 -5237.997,E2 -5237.997} C_VEL
LIN {X 0,Y 517.912,Z 460.286,A -85,B 0,C 180,E1 -5238.555,E2 -5238.555} C_VEL
LIN {X 0,Y 517.617,Z 472.249,A -85,B 0,C 180,E1 -5239.326,E2 -5239.326} C_VEL
LIN {X 0,Y 517.355,Z 482.349,A -85,B 0,C 180,E1 -5240.143,E2 -5240.143} C_VEL
LIN {X 0,Y 517.067,Z 492.042,A -85,B 0,C 180,E1 -5241.112,E2 -5241.112} C_VEL
LIN {X 0,Y 516.828,Z 500.59,A -85,B 0,C 180,E1 -5242.161,E2 -5242.161} C_VEL
LIN {X 0,Y 516.614,Z 509.022,A -85,B 0,C 180,E1 -5243.448,E2 -5243.448} C_VEL
LIN {X 0,Y 516.424,Z 514.858,A -85,B 0,C 180,E1 -5244.566,E2 -5244.566} C_VEL
LIN {X 0,Y 516.315,Z 520.086,A -85,B 0,C 180,E1 -5245.822,E2 -5245.822} C_VEL
LIN {X 0,Y 516.293,Z 524.12,A -85,B 0,C 180,E1 -5247.13,E2 -5247.13} C_VEL
LIN {X 0,Y 516.204,Z 526.993,A -85,B 0,C 180,E1 -5248.458,E2 -5248.458} C_VEL
LIN {X 0,Y 516.225,Z 528.258,A -85,B 0,C 180,E1 -5249.388,E2 -5249.388} C_VEL
LIN {X 0,Y 516.186,Z 528.97,A -85,B 0,C 180,E1 -5250.249,E2 -5250.249} C_VEL
LIN {X 0,Y 516.182,Z 529.177,A -85,B 0,C 180,E1 -5251.157,E2 -5251.157} C_VEL
LIN {X 0,Y 516.182,Z 528.565,A -85,B 0,C 180,E1 -5252.418,E2 -5252.418} C_VEL
LIN {X 0,Y 516.23,Z 526.456,A -85,B 0,C 180,E1 -5253.93,E2 -5253.93} C_VEL
LIN {X 0,Y 516.243,Z 523.408,A -85,B 0,C 180,E1 -5255.231,E2 -5255.231} C_VEL
LIN {X 0,Y 516.37,Z 518.901,A -85,B 0,C 180,E1 -5256.58,E2 -5256.58} C_VEL
LIN {X 0,Y 516.476,Z 513.098,A -85,B 0,C 180,E1 -5257.884,E2 -5257.884} C_VEL
LIN {X 0,Y 516.673,Z 505.849,A -85,B 0,C 180,E1 -5259.163,E2 -5259.163} C_VEL
LIN {X 0,Y 516.841,Z 498.386,A -85,B 0,C 180,E1 -5260.22,E2 -5260.22} C_VEL
LIN {X 0,Y 517.085,Z 489.589,A -85,B 0,C 180,E1 -5261.238,E2 -5261.238} C_VEL
LIN {X 0,Y 517.395,Z 478.818,A -85,B 0,C 180,E1 -5262.251,E2 -5262.251} C_VEL
LIN {X 0,Y 517.579,Z 472.072,A -85,B 0,C 180,E1 -5262.775,E2 -5262.775} C_VEL
LIN {X 0,Y 517.104,Z 467.172,A -85,B 0,C 180,E1 -5263.13,E2 -5263.13} C_VEL
LIN {X 0,Y 514.533,Z 459,A -85,B 0,C 180,E1 -5263.692,E2 -5263.692} C_VEL
LIN {X 0,Y 511.932,Z 450.551,A -85,B 0,C 180,E1 -5264.189,E2 -5264.189} C_VEL
LIN {X 0,Y 511.403,Z 445.115,A -85,B 0,C 180,E1 -5264.436,E2 -5264.436} C_VEL
LIN {X 0,Y 511.386,Z 435.874,A -85,B 0,C 180,E1 -5264.76,E2 -5264.76} C_VEL
LIN {X 0,Y 509.297,Z 424.007,A -85,B 0,C 180,E1 -5265.123,E2 -5265.123} C_VEL
LIN {X 0,Y 509.361,Z 417.212,A -85,B 0,C 180,E1 -5268.165,E2 -5268.165} C_VEL
LIN {X 0,Y 509.432,Z 410.556,A -85,B 0,C 180,E1 -5271.118,E2 -5271.118} C_VEL
LIN {X 0,Y 509.496,Z 404.941,A -85,B 0,C 180,E1 -5273.618,E2 -5273.618} C_VEL
LIN {X 0,Y 509.602,Z 398.386,A -85,B 0,C 180,E1 -5276.519,E2 -5276.519} C_VEL
LIN {X 0,Y 509.636,Z 392.054,A -85,B 0,C 180,E1 -5279.319,E2 -5279.319} C_VEL
LIN {X 0,Y 509.698,Z 384.865,A -85,B 0,C 180,E1 -5282.488,E2 -5282.488} C_VEL
LIN {X 0,Y 509.878,Z 376.976,A -85,B 0,C 180,E1 -5286.006,E2 -5286.006} C_VEL
LIN {X 0,Y 509.849,Z 376.979,A -85,B 0,C 180,E1 -5288.997,E2 -5288.997} C_VEL
LIN {X 0,Y 509.858,Z 376.975,A -85,B 0,C 180,E1 -5291.515,E2 -5291.515} C_VEL
LIN {X 0,Y 509.913,Z 376.968,A -85,B 0,C 180,E1 -5294.817,E2 -5294.817} C_VEL
LIN {X 0,Y 509.902,Z 376.972,A -85,B 0,C 180,E1 -5298.123,E2 -5298.123} C_VEL
LIN {X 0,Y 509.912,Z 376.971,A -85,B 0,C 180,E1 -5301.278,E2 -5301.278} C_VEL
LIN {X 0,Y 509.971,Z 376.965,A -85,B 0,C 180,E1 -5304.463,E2 -5304.463} C_VEL
LIN {X 0,Y 510.043,Z 376.955,A -85,B 0,C 180,E1 -5307.629,E2 -5307.629} C_VEL
LIN {X 0,Y 510.058,Z 377.015,A -85,B 0,C 180,E1 -5310.196,E2 -5310.196} C_VEL
LIN {X 0,Y 509.985,Z 381.152,A -85,B 0,C 180,E1 -5312.368,E2 -5312.368} C_VEL
LIN {X 0,Y 509.791,Z 387.288,A -85,B 0,C 180,E1 -5315.536,E2 -5315.536} C_VEL
LIN {X 0,Y 509.684,Z 391.991,A -85,B 0,C 180,E1 -5317.924,E2 -5317.924} C_VEL
LIN {X 0,Y 509.6,Z 398.334,A -85,B 0,C 180,E1 -5321.13,E2 -5321.13} C_VEL
LIN {X 0,Y 509.475,Z 404.843,A -85,B 0,C 180,E1 -5324.375,E2 -5324.375} C_VEL
LIN {X 0,Y 509.349,Z 411.523,A -85,B 0,C 180,E1 -5327.669,E2 -5327.669} C_VEL
LIN {X 0,Y 509.23,Z 418.484,A -85,B 0,C 180,E1 -5331.026,E2 -5331.026} C_VEL
LIN {X 0,Y 509.266,Z 420.223,A -85,B 0,C 180,E1 -5331.874,E2 -5331.874} C_VEL
LIN {X 0,Y 510.789,Z 431.274,A -85,B 0,C 180,E1 -5332.264,E2 -5332.264} C_VEL
LIN {X 0,Y 510.552,Z 441.879,A -85,B 0,C 180,E1 -5332.738,E2 -5332.738} C_VEL
LIN {X 0,Y 510.256,Z 451.617,A -85,B 0,C 180,E1 -5333.325,E2 -5333.325} C_VEL
LIN {X 0,Y 510.09,Z 460.156,A -85,B 0,C 180,E1 -5333.979,E2 -5333.979} C_VEL
LIN {X 0,Y 509.896,Z 468.372,A -85,B 0,C 180,E1 -5334.762,E2 -5334.762} C_VEL
LIN {X 0,Y 509.661,Z 476.612,A -85,B 0,C 180,E1 -5335.743,E2 -5335.743} C_VEL
LIN {X 0,Y 509.523,Z 483.958,A -85,B 0,C 180,E1 -5336.861,E2 -5336.861} C_VEL
LIN {X 0,Y 509.376,Z 489.664,A -85,B 0,C 180,E1 -5337.991,E2 -5337.991} C_VEL
LIN {X 0,Y 509.304,Z 494.332,A -85,B 0,C 180,E1 -5339.243,E2 -5339.243} C_VEL
LIN {X 0,Y 509.226,Z 497.046,A -85,B 0,C 180,E1 -5340.245,E2 -5340.245} C_VEL
LIN {X 0,Y 509.118,Z 498.765,A -85,B 0,C 180,E1 -5341.145,E2 -5341.145} C_VEL
LIN {X 0,Y 509.103,Z 500.113,A -85,B 0,C 180,E1 -5342.64,E2 -5342.64} C_VEL
LIN {X 0,Y 509.122,Z 499.805,A -85,B 0,C 180,E1 -5344.081,E2 -5344.081} C_VEL
LIN {X 0,Y 509.198,Z 497.867,A -85,B 0,C 180,E1 -5345.48,E2 -5345.48} C_VEL
LIN {X 0,Y 509.252,Z 495.744,A -85,B 0,C 180,E1 -5346.397,E2 -5346.397} C_VEL
LIN {X 0,Y 509.328,Z 492.618,A -85,B 0,C 180,E1 -5347.379,E2 -5347.379} C_VEL
LIN {X 0,Y 509.45,Z 487.243,A -85,B 0,C 180,E1 -5348.623,E2 -5348.623} C_VEL
LIN {X 0,Y 509.573,Z 481.588,A -85,B 0,C 180,E1 -5349.63,E2 -5349.63} C_VEL
LIN {X 0,Y 509.725,Z 475.217,A -85,B 0,C 180,E1 -5350.541,E2 -5350.541} C_VEL
LIN {X 0,Y 509.897,Z 467.659,A -85,B 0,C 180,E1 -5351.418,E2 -5351.418} C_VEL
LIN {X 0,Y 510.169,Z 458.303,A -85,B 0,C 180,E1 -5352.282,E2 -5352.282} C_VEL
LIN {X 0,Y 510.48,Z 447.1,A -85,B 0,C 180,E1 -5353.069,E2 -5353.069} C_VEL
LIN {X 0,Y 510.695,Z 437.087,A -85,B 0,C 180,E1 -5353.595,E2 -5353.595} C_VEL
LIN {X 0,Y 510.533,Z 427.87,A -85,B 0,C 180,E1 -5353.964,E2 -5353.964} C_VEL
LIN {X 0,Y 509.278,Z 420.282,A -85,B 0,C 180,E1 -5354.233,E2 -5354.233} C_VEL
LIN {X 0,Y 509.323,Z 414.592,A -85,B 0,C 180,E1 -5356.994,E2 -5356.994} C_VEL
LIN {X 0,Y 509.365,Z 408.372,A -85,B 0,C 180,E1 -5360.091,E2 -5360.091} C_VEL
LIN {X 0,Y 509.479,Z 402.203,A -85,B 0,C 180,E1 -5363.133,E2 -5363.133} C_VEL
LIN {X 0,Y 509.554,Z 396.809,A -85,B 0,C 180,E1 -5365.842,E2 -5365.842} C_VEL
LIN {X 0,Y 509.654,Z 391.133,A -85,B 0,C 180,E1 -5368.75,E2 -5368.75} C_VEL
LIN {X 0,Y 509.776,Z 386.438,A -85,B 0,C 180,E1 -5371.15,E2 -5371.15} C_VEL
LIN {X 0,Y 509.927,Z 381.252,A -85,B 0,C 180,E1 -5373.83,E2 -5373.83} C_VEL
LIN {X 0,Y 509.902,Z 376.974,A -85,B 0,C 180,E1 -5376.117,E2 -5376.117} C_VEL
LIN {X 0,Y 509.838,Z 376.98,A -85,B 0,C 180,E1 -5378.998,E2 -5378.998} C_VEL
LIN {X 0,Y 509.864,Z 376.98,A -85,B 0,C 180,E1 -5381.998,E2 -5381.998} C_VEL
LIN {X 0,Y 509.885,Z 376.975,A -85,B 0,C 180,E1 -5384.818,E2 -5384.818} C_VEL
LIN {X 0,Y 509.938,Z 376.966,A -85,B 0,C 180,E1 -5388.09,E2 -5388.09} C_VEL
LIN {X 0,Y 509.925,Z 376.971,A -85,B 0,C 180,E1 -5391.28,E2 -5391.28} C_VEL
LIN {X 0,Y 509.99,Z 376.959,A -85,B 0,C 180,E1 -5394.465,E2 -5394.465} C_VEL
LIN {X 0,Y 510.038,Z 376.954,A -85,B 0,C 180,E1 -5397.631,E2 -5397.631} C_VEL
LIN {X 0,Y 510.045,Z 376.953,A -85,B 0,C 180,E1 -5400.79,E2 -5400.79} C_VEL
LIN {X 0,Y 509.963,Z 376.965,A -85,B 0,C 180,E1 -5403.16,E2 -5403.16} C_VEL
LIN {X 0,Y 509.961,Z 376.961,A -85,B 0,C 180,E1 -5406.33,E2 -5406.33} C_VEL
LIN {X 0,Y 509.898,Z 376.972,A -85,B 0,C 180,E1 -5408.721,E2 -5408.721} C_VEL
LIN {X 0,Y 509.93,Z 376.965,A -85,B 0,C 180,E1 -5411.931,E2 -5411.931} C_VEL
LIN {X 0,Y 509.87,Z 376.975,A -85,B 0,C 180,E1 -5415.243,E2 -5415.243} C_VEL
LIN {X 0,Y 509.888,Z 376.973,A -85,B 0,C 180,E1 -5418.01,E2 -5418.01} C_VEL
LIN {X 0,Y 509.839,Z 376.977,A -85,B 0,C 180,E1 -5421.002,E2 -5421.002} C_VEL
LIN {X 0,Y 509.83,Z 376.979,A -85,B 0,C 180,E1 -5423.564,E2 -5423.564} C_VEL
LIN {X 0,Y 509.893,Z 376.97,A -85,B 0,C 180,E1 -5426.381,E2 -5426.381} C_VEL
LIN {X 0,Y 509.865,Z 376.975,A -85,B 0,C 180,E1 -5428.845,E2 -5428.845} C_VEL
LIN {X 0,Y 509.807,Z 376.982,A -85,B 0,C 180,E1 -5431.591,E2 -5431.591} C_VEL
LIN {X 0,Y 509.837,Z 376.979,A -85,B 0,C 180,E1 -5434.415,E2 -5434.415} C_VEL
LIN {X 0,Y 509.802,Z 376.982,A -85,B 0,C 180,E1 -5437.342,E2 -5437.342} C_VEL
LIN {X 0,Y 509.845,Z 376.978,A -85,B 0,C 180,E1 -5440.382,E2 -5440.382} C_VEL
LIN {X 0,Y 509.825,Z 376.981,A -85,B 0,C 180,E1 -5443.066,E2 -5443.066} C_VEL
LIN {X 0,Y 509.816,Z 376.981,A -85,B 0,C 180,E1 -5445.794,E2 -5445.794} C_VEL
LIN {X 0,Y 509.853,Z 376.978,A -85,B 0,C 180,E1 -5448.578,E2 -5448.578} C_VEL
LIN {X 0,Y 509.848,Z 376.978,A -85,B 0,C 180,E1 -5451.665,E2 -5451.665} C_VEL
LIN {X 0,Y 509.837,Z 376.98,A -85,B 0,C 180,E1 -5454.626,E2 -5454.626} C_VEL
LIN {X 0,Y 509.887,Z 377.124,A -85,B 0,C 180,E1 -5456.916,E2 -5456.916} C_VEL
LIN {X 0,Y 511.382,Z 385.264,A -85,B 0,C 180,E1 -5459.439,E2 -5459.439} C_VEL
LIN {X 0,Y 511.371,Z 390.052,A -85,B 0,C 180,E1 -5460.801,E2 -5460.801} C_VEL
LIN {X 0,Y 510.956,Z 399.438,A -85,B 0,C 180,E1 -5463.387,E2 -5463.387} C_VEL
LIN {X 0,Y 510.542,Z 411.089,A -85,B 0,C 180,E1 -5466.474,E2 -5466.474} C_VEL
LIN {X 0,Y 510.15,Z 423.029,A -85,B 0,C 180,E1 -5469.52,E2 -5469.52} C_VEL
LIN {X 0,Y 509.904,Z 436.311,A -85,B 0,C 180,E1 -5472.765,E2 -5472.765} C_VEL
LIN {X 0,Y 509.668,Z 449.36,A -85,B 0,C 180,E1 -5475.936,E2 -5475.936} C_VEL
LIN {X 0,Y 511.465,Z 462.745,A -85,B 0,C 180,E1 -5476.291,E2 -5476.291} C_VEL
LIN {X 0,Y 511.209,Z 475.801,A -85,B 0,C 180,E1 -5476.739,E2 -5476.739} C_VEL
LIN {X 0,Y 510.89,Z 487.234,A -85,B 0,C 180,E1 -5477.287,E2 -5477.287} C_VEL
LIN {X 0,Y 510.556,Z 498.765,A -85,B 0,C 180,E1 -5478.003,E2 -5478.003} C_VEL
LIN {X 0,Y 510.303,Z 509.988,A -85,B 0,C 180,E1 -5478.885,E2 -5478.885} C_VEL
LIN {X 0,Y 509.965,Z 520.1,A -85,B 0,C 180,E1 -5479.882,E2 -5479.882} C_VEL
LIN {X 0,Y 509.698,Z 529.881,A -85,B 0,C 180,E1 -5481.078,E2 -5481.078} C_VEL
LIN {X 0,Y 509.484,Z 537.675,A -85,B 0,C 180,E1 -5482.273,E2 -5482.273} C_VEL
LIN {X 0,Y 509.321,Z 544.837,A -85,B 0,C 180,E1 -5483.664,E2 -5483.664} C_VEL
LIN {X 0,Y 509.247,Z 549.605,A -85,B 0,C 180,E1 -5484.855,E2 -5484.855} C_VEL
LIN {X 0,Y 509.265,Z 553.255,A -85,B 0,C 180,E1 -5486.045,E2 -5486.045} C_VEL
LIN {X 0,Y 509.2,Z 555.132,A -85,B 0,C 180,E1 -5486.837,E2 -5486.837} C_VEL
LIN {X 0,Y 509.19,Z 556.54,A -85,B 0,C 180,E1 -5487.629,E2 -5487.629} C_VEL
LIN {X 0,Y 509.073,Z 558.149,A -85,B 0,C 180,E1 -5489.211,E2 -5489.211} C_VEL
LIN {X 0,Y 509.066,Z 558.368,A -85,B 0,C 180,E1 -5490.002,E2 -5490.002} C_VEL
LIN {X 0,Y 509.113,Z 557.539,A -85,B 0,C 180,E1 -5491.584,E2 -5491.584} C_VEL
LIN {X 0,Y 509.19,Z 556.539,A -85,B 0,C 180,E1 -5492.375,E2 -5492.375} C_VEL
LIN {X 0,Y 509.201,Z 555.132,A -85,B 0,C 180,E1 -5493.166,E2 -5493.166} C_VEL
LIN {X 0,Y 509.219,Z 552.177,A -85,B 0,C 180,E1 -5494.355,E2 -5494.355} C_VEL
LIN {X 0,Y 509.323,Z 548.177,A -85,B 0,C 180,E1 -5495.545,E2 -5495.545} C_VEL
LIN {X 0,Y 509.398,Z 542.461,A -85,B 0,C 180,E1 -5496.846,E2 -5496.846} C_VEL
LIN {X 0,Y 509.539,Z 535.264,A -85,B 0,C 180,E1 -5498.129,E2 -5498.129} C_VEL
LIN {X 0,Y 509.775,Z 526.903,A -85,B 0,C 180,E1 -5499.324,E2 -5499.324} C_VEL
LIN {X 0,Y 510.009,Z 518.296,A -85,B 0,C 180,E1 -5500.321,E2 -5500.321} C_VEL
LIN {X 0,Y 510.399,Z 507.671,A -85,B 0,C 180,E1 -5501.317,E2 -5501.317} C_VEL
LIN {X 0,Y 510.601,Z 496.429,A -85,B 0,C 180,E1 -5502.166,E2 -5502.166} C_VEL
LIN {X 0,Y 510.975,Z 484.465,A -85,B 0,C 180,E1 -5502.866,E2 -5502.866} C_VEL
LIN {X 0,Y 511.306,Z 472.022,A -85,B 0,C 180,E1 -5503.413,E2 -5503.413} C_VEL
LIN {X 0,Y 511.323,Z 460.983,A -85,B 0,C 180,E1 -5503.767,E2 -5503.767} C_VEL
LIN {X 0,Y 509.659,Z 449.373,A -85,B 0,C 180,E1 -5504.068,E2 -5504.068} C_VEL
LIN {X 0,Y 509.849,Z 438.02,A -85,B 0,C 180,E1 -5506.828,E2 -5506.828} C_VEL
LIN {X 0,Y 510.131,Z 426.297,A -85,B 0,C 180,E1 -5509.728,E2 -5509.728} C_VEL
LIN {X 0,Y 510.447,Z 414.496,A -85,B 0,C 180,E1 -5512.708,E2 -5512.708} C_VEL
LIN {X 0,Y 510.829,Z 403.046,A -85,B 0,C 180,E1 -5515.683,E2 -5515.683} C_VEL
LIN {X 0,Y 511.33,Z 391.603,A -85,B 0,C 180,E1 -5518.756,E2 -5518.756} C_VEL
LIN {X 0,Y 511.35,Z 385.139,A -85,B 0,C 180,E1 -5520.567,E2 -5520.567} C_VEL
LIN {X 0,Y 509.874,Z 376.974,A -85,B 0,C 180,E1 -5523.084,E2 -5523.084} C_VEL
LIN {X 0,Y 509.83,Z 376.978,A -85,B 0,C 180,E1 -5525.579,E2 -5525.579} C_VEL
LIN {X 0,Y 509.854,Z 376.979,A -85,B 0,C 180,E1 -5528.339,E2 -5528.339} C_VEL
LIN {X 0,Y 509.808,Z 376.982,A -85,B 0,C 180,E1 -5531.431,E2 -5531.431} C_VEL
LIN {X 0,Y 509.84,Z 376.975,A -85,B 0,C 180,E1 -5534.671,E2 -5534.671} C_VEL
LIN {X 0,Y 509.807,Z 376.981,A -85,B 0,C 180,E1 -5537.507,E2 -5537.507} C_VEL
LIN {X 0,Y 509.843,Z 376.979,A -85,B 0,C 180,E1 -5540.647,E2 -5540.647} C_VEL
LIN {X 0,Y 509.83,Z 376.976,A -85,B 0,C 180,E1 -5543.647,E2 -5543.647} C_VEL
LIN {X 0,Y 509.847,Z 376.976,A -85,B 0,C 180,E1 -5546.538,E2 -5546.538} C_VEL
LIN {X 0,Y 509.839,Z 376.977,A -85,B 0,C 180,E1 -5549.333,E2 -5549.333} C_VEL
LIN {X 0,Y 509.832,Z 376.977,A -85,B 0,C 180,E1 -5552.051,E2 -5552.051} C_VEL
LIN {X 0,Y 509.785,Z 376.984,A -85,B 0,C 180,E1 -5554.699,E2 -5554.699} C_VEL
LIN {X 0,Y 509.829,Z 376.977,A -85,B 0,C 180,E1 -5557.459,E2 -5557.459} C_VEL
LIN {X 0,Y 509.92,Z 376.966,A -85,B 0,C 180,E1 -5559.845,E2 -5559.845} C_VEL
LIN {X 0,Y 509.886,Z 376.97,A -85,B 0,C 180,E1 -5563.175,E2 -5563.175} C_VEL
LIN {X 0,Y 509.866,Z 376.977,A -85,B 0,C 180,E1 -5565.634,E2 -5565.634} C_VEL
LIN {X 0,Y 509.91,Z 376.968,A -85,B 0,C 180,E1 -5568.874,E2 -5568.874} C_VEL
LIN {X 0,Y 509.877,Z 376.971,A -85,B 0,C 180,E1 -5572.077,E2 -5572.077} C_VEL
LIN {X 0,Y 509.95,Z 376.965,A -85,B 0,C 180,E1 -5574.464,E2 -5574.464} C_VEL
LIN {X 0,Y 509.599,Z 377.105,A -85,B 0,C 180,E1 -5577.085,E2 -5577.085} C_VEL
LIN {X 0,Y 509.799,Z 384.416,A -85,B 0,C 180,E1 -5580,E2 -5580} C_VEL
LIN {X 0,Y 509.538,Z 390.292,A -85,B 0,C 180,E1 -5582.371,E2 -5582.371} C_VEL
LIN {X 0,Y 509.618,Z 395.977,A -85,B 0,C 180,E1 -5584.746,E2 -5584.746} C_VEL
LIN {X 0,Y 509.573,Z 401.554,A -85,B 0,C 180,E1 -5587.13,E2 -5587.13} C_VEL
LIN {X 0,Y 509.481,Z 407.114,A -85,B 0,C 180,E1 -5589.528,E2 -5589.528} C_VEL
LIN {X 0,Y 509.457,Z 412.757,A -85,B 0,C 180,E1 -5591.942,E2 -5591.942} C_VEL
LIN {X 0,Y 509.366,Z 420.175,A -85,B 0,C 180,E1 -5595.198,E2 -5595.198} C_VEL
LIN {X 0,Y 509.283,Z 424.201,A -85,B 0,C 180,E1 -5596.975,E2 -5596.975} C_VEL
LIN {X 0,Y 511.561,Z 436.714,A -85,B 0,C 180,E1 -5597.36,E2 -5597.36} C_VEL
LIN {X 0,Y 511.307,Z 448.802,A -85,B 0,C 180,E1 -5597.804,E2 -5597.804} C_VEL
LIN {X 0,Y 510.949,Z 461.396,A -85,B 0,C 180,E1 -5598.443,E2 -5598.443} C_VEL
LIN {X 0,Y 510.654,Z 472.605,A -85,B 0,C 180,E1 -5599.183,E2 -5599.183} C_VEL
LIN {X 0,Y 510.35,Z 482.921,A -85,B 0,C 180,E1 -5600.032,E2 -5600.032} C_VEL
LIN {X 0,Y 510.048,Z 492.349,A -85,B 0,C 180,E1 -5600.993,E2 -5600.993} C_VEL
LIN {X 0,Y 509.802,Z 500.757,A -85,B 0,C 180,E1 -5602.04,E2 -5602.04} C_VEL
LIN {X 0,Y 509.578,Z 508.035,A -85,B 0,C 180,E1 -5603.145,E2 -5603.145} C_VEL
LIN {X 0,Y 509.362,Z 514.955,A -85,B 0,C 180,E1 -5604.452,E2 -5604.452} C_VEL
LIN {X 0,Y 509.233,Z 520.324,A -85,B 0,C 180,E1 -5605.768,E2 -5605.768} C_VEL
LIN {X 0,Y 509.219,Z 524.369,A -85,B 0,C 180,E1 -5607.094,E2 -5607.094} C_VEL
LIN {X 0,Y 509.133,Z 526.417,A -85,B 0,C 180,E1 -5607.991,E2 -5607.991} C_VEL
LIN {X 0,Y 509.119,Z 528.684,A -85,B 0,C 180,E1 -5609.579,E2 -5609.579} C_VEL
LIN {X 0,Y 509.105,Z 529.37,A -85,B 0,C 180,E1 -5611.141,E2 -5611.141} C_VEL
LIN {X 0,Y 509.08,Z 528.557,A -85,B 0,C 180,E1 -5612.634,E2 -5612.634} C_VEL
LIN {X 0,Y 509.136,Z 526.437,A -85,B 0,C 180,E1 -5614.082,E2 -5614.082} C_VEL
LIN {X 0,Y 509.188,Z 523.046,A -85,B 0,C 180,E1 -5615.477,E2 -5615.477} C_VEL
LIN {X 0,Y 509.323,Z 518.349,A -85,B 0,C 180,E1 -5616.838,E2 -5616.838} C_VEL
LIN {X 0,Y 509.43,Z 512.4,A -85,B 0,C 180,E1 -5618.152,E2 -5618.152} C_VEL
LIN {X 0,Y 509.64,Z 504.907,A -85,B 0,C 180,E1 -5619.443,E2 -5619.443} C_VEL
LIN {X 0,Y 509.894,Z 496.942,A -85,B 0,C 180,E1 -5620.544,E2 -5620.544} C_VEL
LIN {X 0,Y 510.134,Z 488.192,A -85,B 0,C 180,E1 -5621.539,E2 -5621.539} C_VEL
LIN {X 0,Y 510.441,Z 478.672,A -85,B 0,C 180,E1 -5622.427,E2 -5622.427} C_VEL
LIN {X 0,Y 510.737,Z 467.245,A -85,B 0,C 180,E1 -5623.281,E2 -5623.281} C_VEL
LIN {X 0,Y 511.066,Z 455.224,A -85,B 0,C 180,E1 -5623.984,E2 -5623.984} C_VEL
LIN {X 0,Y 511.403,Z 445.115,A -85,B 0,C 180,E1 -5624.436,E2 -5624.436} C_VEL
LIN {X 0,Y 510.753,Z 441.501,A -85,B 0,C 180,E1 -5624.594,E2 -5624.594} C_VEL
LIN {X 0,Y 507.68,Z 436.08,A -85,B 0,C 180,E1 -5624.866,E2 -5624.866} C_VEL
LIN {X 0,Y 504.124,Z 430.655,A -85,B 0,C 180,E1 -5625.116,E2 -5625.116} C_VEL
LIN {X 0,Y 502.752,Z 426.988,A -85,B 0,C 180,E1 -5625.237,E2 -5625.237} C_VEL
LIN {X 0,Y 502.254,Z 424.203,A -85,B 0,C 180,E1 -5625.314,E2 -5625.314} C_VEL
LIN {X 0,Y 502.308,Z 417.37,A -85,B 0,C 180,E1 -5628.377,E2 -5628.377} C_VEL
LIN {X 0,Y 502.371,Z 411.532,A -85,B 0,C 180,E1 -5630.983,E2 -5630.983} C_VEL
LIN {X 0,Y 502.466,Z 404.304,A -85,B 0,C 180,E1 -5634.217,E2 -5634.217} C_VEL
LIN {X 0,Y 502.543,Z 397.965,A -85,B 0,C 180,E1 -5637.044,E2 -5637.044} C_VEL
LIN {X 0,Y 502.628,Z 391.118,A -85,B 0,C 180,E1 -5640.102,E2 -5640.102} C_VEL
LIN {X 0,Y 502.651,Z 383.632,A -85,B 0,C 180,E1 -5643.42,E2 -5643.42} C_VEL
LIN {X 0,Y 502.838,Z 377.853,A -85,B 0,C 180,E1 -5645.978,E2 -5645.978} C_VEL
LIN {X 0,Y 502.832,Z 377.85,A -85,B 0,C 180,E1 -5649.463,E2 -5649.463} C_VEL
LIN {X 0,Y 502.819,Z 377.855,A -85,B 0,C 180,E1 -5652.09,E2 -5652.09} C_VEL
LIN {X 0,Y 502.847,Z 377.85,A -85,B 0,C 180,E1 -5655.428,E2 -5655.428} C_VEL
LIN {X 0,Y 502.877,Z 377.845,A -85,B 0,C 180,E1 -5658.715,E2 -5658.715} C_VEL
LIN {X 0,Y 502.902,Z 377.841,A -85,B 0,C 180,E1 -5661.965,E2 -5661.965} C_VEL
LIN {X 0,Y 502.925,Z 377.842,A -85,B 0,C 180,E1 -5664.385,E2 -5664.385} C_VEL
LIN {X 0,Y 503.011,Z 377.831,A -85,B 0,C 180,E1 -5667.596,E2 -5667.596} C_VEL
LIN {X 0,Y 503.03,Z 378.002,A -85,B 0,C 180,E1 -5670.198,E2 -5670.198} C_VEL
LIN {X 0,Y 502.93,Z 382.16,A -85,B 0,C 180,E1 -5672.401,E2 -5672.401} C_VEL
LIN {X 0,Y 502.749,Z 388.336,A -85,B 0,C 180,E1 -5675.614,E2 -5675.614} C_VEL
LIN {X 0,Y 502.629,Z 393.038,A -85,B 0,C 180,E1 -5678.036,E2 -5678.036} C_VEL
LIN {X 0,Y 502.532,Z 399.427,A -85,B 0,C 180,E1 -5681.289,E2 -5681.289} C_VEL
LIN {X 0,Y 502.399,Z 405.984,A -85,B 0,C 180,E1 -5684.582,E2 -5684.582} C_VEL
LIN {X 0,Y 502.25,Z 412.679,A -85,B 0,C 180,E1 -5687.914,E2 -5687.914} C_VEL
LIN {X 0,Y 502.184,Z 417.934,A -85,B 0,C 180,E1 -5690.477,E2 -5690.477} C_VEL
LIN {X 0,Y 502.192,Z 420.613,A -85,B 0,C 180,E1 -5691.712,E2 -5691.712} C_VEL
LIN {X 0,Y 503.773,Z 430.909,A -85,B 0,C 180,E1 -5692.071,E2 -5692.071} C_VEL
LIN {X 0,Y 503.593,Z 441.696,A -85,B 0,C 180,E1 -5692.554,E2 -5692.554} C_VEL
LIN {X 0,Y 503.32,Z 451.165,A -85,B 0,C 180,E1 -5693.121,E2 -5693.121} C_VEL
LIN {X 0,Y 503.093,Z 461.122,A -85,B 0,C 180,E1 -5693.896,E2 -5693.896} C_VEL
LIN {X 0,Y 502.87,Z 470.117,A -85,B 0,C 180,E1 -5694.786,E2 -5694.786} C_VEL
LIN {X 0,Y 502.646,Z 477.349,A -85,B 0,C 180,E1 -5695.684,E2 -5695.684} C_VEL
LIN {X 0,Y 502.474,Z 484.56,A -85,B 0,C 180,E1 -5696.81,E2 -5696.81} C_VEL
LIN {X 0,Y 502.348,Z 489.672,A -85,B 0,C 180,E1 -5697.83,E2 -5697.83} C_VEL
LIN {X 0,Y 502.247,Z 493.722,A -85,B 0,C 180,E1 -5698.863,E2 -5698.863} C_VEL
LIN {X 0,Y 502.139,Z 497.56,A -85,B 0,C 180,E1 -5700.253,E2 -5700.253} C_VEL
LIN {X 0,Y 502.026,Z 499.488,A -85,B 0,C 180,E1 -5701.356,E2 -5701.356} C_VEL
LIN {X 0,Y 502.03,Z 500.287,A -85,B 0,C 180,E1 -5702.136,E2 -5702.136} C_VEL
LIN {X 0,Y 502.016,Z 500.623,A -85,B 0,C 180,E1 -5703.089,E2 -5703.089} C_VEL
LIN {X 0,Y 502.05,Z 500.001,A -85,B 0,C 180,E1 -5704.319,E2 -5704.319} C_VEL
LIN {X 0,Y 502.068,Z 499.127,A -85,B 0,C 180,E1 -5705.021,E2 -5705.021} C_VEL
LIN {X 0,Y 502.193,Z 496.025,A -85,B 0,C 180,E1 -5706.493,E2 -5706.493} C_VEL
LIN {X 0,Y 502.285,Z 492.779,A -85,B 0,C 180,E1 -5707.511,E2 -5707.511} C_VEL
LIN {X 0,Y 502.413,Z 487.768,A -85,B 0,C 180,E1 -5708.682,E2 -5708.682} C_VEL
LIN {X 0,Y 502.529,Z 482.061,A -85,B 0,C 180,E1 -5709.719,E2 -5709.719} C_VEL
LIN {X 0,Y 502.749,Z 474.749,A -85,B 0,C 180,E1 -5710.768,E2 -5710.768} C_VEL
LIN {X 0,Y 502.979,Z 466.431,A -85,B 0,C 180,E1 -5711.713,E2 -5711.713} C_VEL
LIN {X 0,Y 503.261,Z 457.239,A -85,B 0,C 180,E1 -5712.537,E2 -5712.537} C_VEL
LIN {X 0,Y 503.525,Z 447.324,A -85,B 0,C 180,E1 -5713.232,E2 -5713.232} C_VEL
LIN {X 0,Y 503.774,Z 437.318,A -85,B 0,C 180,E1 -5713.762,E2 -5713.762} C_VEL
LIN {X 0,Y 503.583,Z 428.598,A -85,B 0,C 180,E1 -5714.12,E2 -5714.12} C_VEL
LIN {X 0,Y 502.2,Z 420.565,A -85,B 0,C 180,E1 -5714.401,E2 -5714.401} C_VEL
LIN {X 0,Y 502.257,Z 414.758,A -85,B 0,C 180,E1 -5717.262,E2 -5717.262} C_VEL
LIN {X 0,Y 502.321,Z 408.661,A -85,B 0,C 180,E1 -5720.305,E2 -5720.305} C_VEL
LIN {X 0,Y 502.438,Z 403.207,A -85,B 0,C 180,E1 -5723.025,E2 -5723.025} C_VEL
LIN {X 0,Y 502.503,Z 397.422,A -85,B 0,C 180,E1 -5725.983,E2 -5725.983} C_VEL
LIN {X 0,Y 502.616,Z 391.837,A -85,B 0,C 180,E1 -5728.845,E2 -5728.845} C_VEL
LIN {X 0,Y 502.771,Z 386.296,A -85,B 0,C 180,E1 -5731.714,E2 -5731.714} C_VEL
LIN {X 0,Y 502.884,Z 381.298,A -85,B 0,C 180,E1 -5734.327,E2 -5734.327} C_VEL
LIN {X 0,Y 502.856,Z 377.852,A -85,B 0,C 180,E1 -5736.199,E2 -5736.199} C_VEL
LIN {X 0,Y 502.829,Z 377.854,A -85,B 0,C 180,E1 -5739.548,E2 -5739.548} C_VEL
LIN {X 0,Y 502.838,Z 377.855,A -85,B 0,C 180,E1 -5742.092,E2 -5742.092} C_VEL
LIN {X 0,Y 502.83,Z 377.852,A -85,B 0,C 180,E1 -5745.429,E2 -5745.429} C_VEL
LIN {X 0,Y 502.883,Z 377.847,A -85,B 0,C 180,E1 -5748.717,E2 -5748.717} C_VEL
LIN {X 0,Y 502.881,Z 377.844,A -85,B 0,C 180,E1 -5751.967,E2 -5751.967} C_VEL
LIN {X 0,Y 502.942,Z 377.838,A -85,B 0,C 180,E1 -5754.387,E2 -5754.387} C_VEL
LIN {X 0,Y 503.009,Z 377.83,A -85,B 0,C 180,E1 -5757.598,E2 -5757.598} C_VEL
LIN {X 0,Y 503.015,Z 377.828,A -85,B 0,C 180,E1 -5760.801,E2 -5760.801} C_VEL
LIN {X 0,Y 502.905,Z 377.844,A -85,B 0,C 180,E1 -5763.205,E2 -5763.205} C_VEL
LIN {X 0,Y 502.909,Z 377.839,A -85,B 0,C 180,E1 -5766.419,E2 -5766.419} C_VEL
LIN {X 0,Y 502.857,Z 377.848,A -85,B 0,C 180,E1 -5768.844,E2 -5768.844} C_VEL
LIN {X 0,Y 502.872,Z 377.845,A -85,B 0,C 180,E1 -5772.101,E2 -5772.101} C_VEL
LIN {X 0,Y 502.826,Z 377.852,A -85,B 0,C 180,E1 -5775.401,E2 -5775.401} C_VEL
LIN {X 0,Y 502.841,Z 377.85,A -85,B 0,C 180,E1 -5778.13,E2 -5778.13} C_VEL
LIN {X 0,Y 502.779,Z 377.855,A -85,B 0,C 180,E1 -5781.312,E2 -5781.312} C_VEL
LIN {X 0,Y 502.781,Z 377.855,A -85,B 0,C 180,E1 -5783.915,E2 -5783.915} C_VEL
LIN {X 0,Y 502.86,Z 377.846,A -85,B 0,C 180,E1 -5786.567,E2 -5786.567} C_VEL
LIN {X 0,Y 502.819,Z 377.851,A -85,B 0,C 180,E1 -5789.288,E2 -5789.288} C_VEL
LIN {X 0,Y 502.769,Z 377.857,A -85,B 0,C 180,E1 -5792.086,E2 -5792.086} C_VEL
LIN {X 0,Y 502.792,Z 377.856,A -85,B 0,C 180,E1 -5794.967,E2 -5794.967} C_VEL
LIN {X 0,Y 502.78,Z 377.86,A -85,B 0,C 180,E1 -5797.955,E2 -5797.955} C_VEL
LIN {X 0,Y 502.811,Z 377.854,A -85,B 0,C 180,E1 -5801.067,E2 -5801.067} C_VEL
LIN {X 0,Y 502.768,Z 377.862,A -85,B 0,C 180,E1 -5803.378,E2 -5803.378} C_VEL
LIN {X 0,Y 502.775,Z 377.857,A -85,B 0,C 180,E1 -5805.663,E2 -5805.663} C_VEL
LIN {X 0,Y 502.817,Z 377.853,A -85,B 0,C 180,E1 -5807.866,E2 -5807.866} C_VEL
LIN {X 0,Y 502.81,Z 377.855,A -85,B 0,C 180,E1 -5811.028,E2 -5811.028} C_VEL
LIN {X 0,Y 502.776,Z 377.861,A -85,B 0,C 180,E1 -5814.169,E2 -5814.169} C_VEL
LIN {X 0,Y 502.825,Z 377.918,A -85,B 0,C 180,E1 -5816.613,E2 -5816.613} C_VEL
LIN {X 0,Y 504.452,Z 386.725,A -85,B 0,C 180,E1 -5819.401,E2 -5819.401} C_VEL
LIN {X 0,Y 504.326,Z 393.642,A -85,B 0,C 180,E1 -5821.394,E2 -5821.394} C_VEL
LIN {X 0,Y 503.792,Z 404.468,A -85,B 0,C 180,E1 -5824.379,E2 -5824.379} C_VEL
LIN {X 0,Y 503.426,Z 414.751,A -85,B 0,C 180,E1 -5827.13,E2 -5827.13} C_VEL
LIN {X 0,Y 503.071,Z 425.891,A -85,B 0,C 180,E1 -5829.987,E2 -5829.987} C_VEL
LIN {X 0,Y 502.808,Z 437.682,A -85,B 0,C 180,E1 -5832.933,E2 -5832.933} C_VEL
LIN {X 0,Y 502.602,Z 449.13,A -85,B 0,C 180,E1 -5835.76,E2 -5835.76} C_VEL
LIN {X 0,Y 504.53,Z 463.582,A -85,B 0,C 180,E1 -5836.15,E2 -5836.15} C_VEL
LIN {X 0,Y 504.242,Z 476.206,A -85,B 0,C 180,E1 -5836.604,E2 -5836.604} C_VEL
LIN {X 0,Y 503.889,Z 488.36,A -85,B 0,C 180,E1 -5837.209,E2 -5837.209} C_VEL
LIN {X 0,Y 503.527,Z 499.365,A -85,B 0,C 180,E1 -5837.917,E2 -5837.917} C_VEL
LIN {X 0,Y 503.259,Z 510.562,A -85,B 0,C 180,E1 -5838.83,E2 -5838.83} C_VEL
LIN {X 0,Y 502.91,Z 519.609,A -85,B 0,C 180,E1 -5839.738,E2 -5839.738} C_VEL
LIN {X 0,Y 502.648,Z 529.413,A -85,B 0,C 180,E1 -5840.952,E2 -5840.952} C_VEL
LIN {X 0,Y 502.404,Z 537.229,A -85,B 0,C 180,E1 -5842.163,E2 -5842.163} C_VEL
LIN {X 0,Y 502.226,Z 544.032,A -85,B 0,C 180,E1 -5843.493,E2 -5843.493} C_VEL
LIN {X 0,Y 502.182,Z 549.182,A -85,B 0,C 180,E1 -5844.783,E2 -5844.783} C_VEL
LIN {X 0,Y 502.16,Z 552.837,A -85,B 0,C 180,E1 -5845.989,E2 -5845.989} C_VEL
LIN {X 0,Y 502.121,Z 554.72,A -85,B 0,C 180,E1 -5846.792,E2 -5846.792} C_VEL
LIN {X 0,Y 502.12,Z 556.132,A -85,B 0,C 180,E1 -5847.595,E2 -5847.595} C_VEL
LIN {X 0,Y 501.99,Z 557.744,A -85,B 0,C 180,E1 -5849.2,E2 -5849.2} C_VEL
LIN {X 0,Y 501.981,Z 557.963,A -85,B 0,C 180,E1 -5850.002,E2 -5850.002} C_VEL
LIN {X 0,Y 502.037,Z 557.135,A -85,B 0,C 180,E1 -5851.606,E2 -5851.606} C_VEL
LIN {X 0,Y 502.121,Z 556.137,A -85,B 0,C 180,E1 -5852.408,E2 -5852.408} C_VEL
LIN {X 0,Y 502.122,Z 554.727,A -85,B 0,C 180,E1 -5853.211,E2 -5853.211} C_VEL
LIN {X 0,Y 502.115,Z 551.768,A -85,B 0,C 180,E1 -5854.417,E2 -5854.417} C_VEL
LIN {X 0,Y 502.24,Z 547.764,A -85,B 0,C 180,E1 -5855.623,E2 -5855.623} C_VEL
LIN {X 0,Y 502.333,Z 541.683,A -85,B 0,C 180,E1 -5857.013,E2 -5857.013} C_VEL
LIN {X 0,Y 502.485,Z 534.831,A -85,B 0,C 180,E1 -5858.244,E2 -5858.244} C_VEL
LIN {X 0,Y 502.724,Z 526.455,A -85,B 0,C 180,E1 -5859.456,E2 -5859.456} C_VEL
LIN {X 0,Y 502.995,Z 517.821,A -85,B 0,C 180,E1 -5860.467,E2 -5860.467} C_VEL
LIN {X 0,Y 503.395,Z 507.167,A -85,B 0,C 180,E1 -5861.477,E2 -5861.477} C_VEL
LIN {X 0,Y 503.59,Z 496.815,A -85,B 0,C 180,E1 -5862.272,E2 -5862.272} C_VEL
LIN {X 0,Y 504.001,Z 484.829,A -85,B 0,C 180,E1 -5862.996,E2 -5862.996} C_VEL
LIN {X 0,Y 504.328,Z 472.583,A -85,B 0,C 180,E1 -5863.551,E2 -5863.551} C_VEL
LIN {X 0,Y 504.387,Z 461.886,A -85,B 0,C 180,E1 -5863.909,E2 -5863.909} C_VEL
LIN {X 0,Y 502.678,Z 450.088,A -85,B 0,C 180,E1 -5864.215,E2 -5864.215} C_VEL
LIN {X 0,Y 502.601,Z 449.168,A -85,B 0,C 180,E1 -5864.243,E2 -5864.243} C_VEL
LIN {X 0,Y 502.809,Z 437.806,A -85,B 0,C 180,E1 -5867.071,E2 -5867.071} C_VEL
LIN {X 0,Y 503.104,Z 426.094,A -85,B 0,C 180,E1 -5870.015,E2 -5870.015} C_VEL
LIN {X 0,Y 503.477,Z 414.468,A -85,B 0,C 180,E1 -5873.009,E2 -5873.009} C_VEL
LIN {X 0,Y 503.903,Z 402.945,A -85,B 0,C 180,E1 -5876.063,E2 -5876.063} C_VEL
LIN {X 0,Y 504.438,Z 391.569,A -85,B 0,C 180,E1 -5879.186,E2 -5879.186} C_VEL
LIN {X 0,Y 504.419,Z 386.608,A -85,B 0,C 180,E1 -5880.6,E2 -5880.6} C_VEL
LIN {X 0,Y 502.843,Z 377.85,A -85,B 0,C 180,E1 -5883.33,E2 -5883.33} C_VEL
LIN {X 0,Y 502.775,Z 377.859,A -85,B 0,C 180,E1 -5885.952,E2 -5885.952} C_VEL
LIN {X 0,Y 502.799,Z 377.853,A -85,B 0,C 180,E1 -5888.977,E2 -5888.977} C_VEL
LIN {X 0,Y 502.75,Z 377.861,A -85,B 0,C 180,E1 -5892.192,E2 -5892.192} C_VEL
LIN {X 0,Y 502.791,Z 377.856,A -85,B 0,C 180,E1 -5895.471,E2 -5895.471} C_VEL
LIN {X 0,Y 502.777,Z 377.857,A -85,B 0,C 180,E1 -5898.929,E2 -5898.929} C_VEL
LIN {X 0,Y 502.798,Z 377.851,A -85,B 0,C 180,E1 -5902.046,E2 -5902.046} C_VEL
LIN {X 0,Y 502.801,Z 377.852,A -85,B 0,C 180,E1 -5905.034,E2 -5905.034} C_VEL
LIN {X 0,Y 502.787,Z 377.859,A -85,B 0,C 180,E1 -5907.915,E2 -5907.915} C_VEL
LIN {X 0,Y 502.808,Z 377.85,A -85,B 0,C 180,E1 -5910.711,E2 -5910.711} C_VEL
LIN {X 0,Y 502.774,Z 377.86,A -85,B 0,C 180,E1 -5913.461,E2 -5913.461} C_VEL
LIN {X 0,Y 502.76,Z 377.856,A -85,B 0,C 180,E1 -5916.084,E2 -5916.084} C_VEL
LIN {X 0,Y 502.786,Z 377.859,A -85,B 0,C 180,E1 -5918.689,E2 -5918.689} C_VEL
LIN {X 0,Y 502.834,Z 377.848,A -85,B 0,C 180,E1 -5921.248,E2 -5921.248} C_VEL
LIN {X 0,Y 502.826,Z 377.853,A -85,B 0,C 180,E1 -5923.767,E2 -5923.767} C_VEL
LIN {X 0,Y 502.831,Z 377.851,A -85,B 0,C 180,E1 -5926.254,E2 -5926.254} C_VEL
LIN {X 0,Y 502.876,Z 377.844,A -85,B 0,C 180,E1 -5928.717,E2 -5928.717} C_VEL
LIN {X 0,Y 502.849,Z 377.847,A -85,B 0,C 180,E1 -5931.966,E2 -5931.966} C_VEL
LIN {X 0,Y 502.905,Z 377.842,A -85,B 0,C 180,E1 -5934.386,E2 -5934.386} C_VEL
LIN {X 0,Y 502.57,Z 378.042,A -85,B 0,C 180,E1 -5937.094,E2 -5937.094} C_VEL
LIN {X 0,Y 502.759,Z 385.284,A -85,B 0,C 180,E1 -5940,E2 -5940} C_VEL
LIN {X 0,Y 502.486,Z 393.107,A -85,B 0,C 180,E1 -5943.207,E2 -5943.207} C_VEL
LIN {X 0,Y 502.526,Z 398.761,A -85,B 0,C 180,E1 -5945.618,E2 -5945.618} C_VEL
LIN {X 0,Y 502.496,Z 404.456,A -85,B 0,C 180,E1 -5948.04,E2 -5948.04} C_VEL
LIN {X 0,Y 502.429,Z 411.951,A -85,B 0,C 180,E1 -5951.293,E2 -5951.293} C_VEL
LIN {X 0,Y 502.317,Z 419.442,A -85,B 0,C 180,E1 -5954.586,E2 -5954.586} C_VEL
LIN {X 0,Y 502.216,Z 424.377,A -85,B 0,C 180,E1 -5956.775,E2 -5956.775} C_VEL
LIN {X 0,Y 504.609,Z 437.416,A -85,B 0,C 180,E1 -5957.189,E2 -5957.189} C_VEL
LIN {X 0,Y 504.397,Z 449.353,A -85,B 0,C 180,E1 -5957.641,E2 -5957.641} C_VEL
LIN {X 0,Y 504.008,Z 461.668,A -85,B 0,C 180,E1 -5958.277,E2 -5958.277} C_VEL
LIN {X 0,Y 503.679,Z 472.973,A -85,B 0,C 180,E1 -5959.036,E2 -5959.036} C_VEL
LIN {X 0,Y 503.355,Z 483.256,A -85,B 0,C 180,E1 -5959.897,E2 -5959.897} C_VEL
LIN {X 0,Y 503.043,Z 493.009,A -85,B 0,C 180,E1 -5960.912,E2 -5960.912} C_VEL
LIN {X 0,Y 502.761,Z 501.233,A -85,B 0,C 180,E1 -5961.958,E2 -5961.958} C_VEL
LIN {X 0,Y 502.526,Z 508.316,A -85,B 0,C 180,E1 -5963.053,E2 -5963.053} C_VEL
LIN {X 0,Y 502.328,Z 514.613,A -85,B 0,C 180,E1 -5964.248,E2 -5964.248} C_VEL
LIN {X 0,Y 502.22,Z 518.931,A -85,B 0,C 180,E1 -5965.265,E2 -5965.265} C_VEL
LIN {X 0,Y 502.146,Z 523.419,A -85,B 0,C 180,E1 -5966.607,E2 -5966.607} C_VEL
LIN {X 0,Y 502.039,Z 526.919,A -85,B 0,C 180,E1 -5968.123,E2 -5968.123} C_VEL
LIN {X 0,Y 502.015,Z 529.081,A -85,B 0,C 180,E1 -5969.775,E2 -5969.775} C_VEL
LIN {X 0,Y 501.995,Z 529.519,A -85,B 0,C 180,E1 -5971.349,E2 -5971.349} C_VEL
LIN {X 0,Y 502.008,Z 528.543,A -85,B 0,C 180,E1 -5972.86,E2 -5972.86} C_VEL
LIN {X 0,Y 502.074,Z 526.222,A -85,B 0,C 180,E1 -5974.321,E2 -5974.321} C_VEL
LIN {X 0,Y 502.133,Z 522.648,A -85,B 0,C 180,E1 -5975.728,E2 -5975.728} C_VEL
LIN {X 0,Y 502.285,Z 517.796,A -85,B 0,C 180,E1 -5977.102,E2 -5977.102} C_VEL
LIN {X 0,Y 502.418,Z 511.634,A -85,B 0,C 180,E1 -5978.431,E2 -5978.431} C_VEL
LIN {X 0,Y 502.632,Z 503.934,A -85,B 0,C 180,E1 -5979.732,E2 -5979.732} C_VEL
LIN {X 0,Y 502.906,Z 496.339,A -85,B 0,C 180,E1 -5980.771,E2 -5980.771} C_VEL
LIN {X 0,Y 503.222,Z 486.953,A -85,B 0,C 180,E1 -5981.826,E2 -5981.826} C_VEL
LIN {X 0,Y 503.554,Z 476.409,A -85,B 0,C 180,E1 -5982.78,E2 -5982.78} C_VEL
LIN {X 0,Y 503.888,Z 465.177,A -85,B 0,C 180,E1 -5983.595,E2 -5983.595} C_VEL
LIN {X 0,Y 504.245,Z 452.685,A -85,B 0,C 180,E1 -5984.291,E2 -5984.291} C_VEL
LIN {X 0,Y 504.577,Z 439.536,A -85,B 0,C 180,E1 -5984.832,E2 -5984.832} C_VEL
LIN {X 0,Y 504.258,Z 435.181,A -85,B 0,C 180,E1 -5984.98,E2 -5984.98} C_VEL
LIN {X 0,Y 502.752,Z 426.988,A -85,B 0,C 180,E1 -5985.237,E2 -5985.237} C_VEL
LIN {X 0,Y 502.051,Z 425.112,A -85,B 0,C 180,E1 -5985.37,E2 -5985.37} C_VEL
LIN {X 0,Y 500.841,Z 423.613,A -85,B 0,C 180,E1 -5985.671,E2 -5985.671} C_VEL
LIN {X 0,Y 498.115,Z 421.778,A -85,B 0,C 180,E1 -5986.561,E2 -5986.561} C_VEL
LIN {X 0,Y 496.053,Z 419.944,A -85,B 0,C 180,E1 -5987.564,E2 -5987.564} C_VEL
LIN {X 0,Y 495.25,Z 417.559,A -85,B 0,C 180,E1 -5988.579,E2 -5988.579} C_VEL
LIN {X 0,Y 495.319,Z 411.36,A -85,B 0,C 180,E1 -5991.367,E2 -5991.367} C_VEL
LIN {X 0,Y 495.4,Z 404.559,A -85,B 0,C 180,E1 -5994.432,E2 -5994.432} C_VEL
LIN {X 0,Y 495.492,Z 399.274,A -85,B 0,C 180,E1 -5996.808,E2 -5996.808} C_VEL
LIN {X 0,Y 495.575,Z 392.388,A -85,B 0,C 180,E1 -5999.89,E2 -5999.89} C_VEL
LIN {X 0,Y 495.604,Z 385.406,A -85,B 0,C 180,E1 -6003.012,E2 -6003.012} C_VEL
LIN {X 0,Y 495.782,Z 378.731,A -85,B 0,C 180,E1 -6006.059,E2 -6006.059} C_VEL
LIN {X 0,Y 495.781,Z 378.729,A -85,B 0,C 180,E1 -6009.323,E2 -6009.323} C_VEL
LIN {X 0,Y 495.781,Z 378.731,A -85,B 0,C 180,E1 -6011.827,E2 -6011.827} C_VEL
LIN {X 0,Y 495.826,Z 378.722,A -85,B 0,C 180,E1 -6014.547,E2 -6014.547} C_VEL
LIN {X 0,Y 495.83,Z 378.723,A -85,B 0,C 180,E1 -6017.964,E2 -6017.964} C_VEL
LIN {X 0,Y 495.839,Z 378.722,A -85,B 0,C 180,E1 -6021.029,E2 -6021.029} C_VEL
LIN {X 0,Y 495.88,Z 378.719,A -85,B 0,C 180,E1 -6024.305,E2 -6024.305} C_VEL
LIN {X 0,Y 495.977,Z 378.706,A -85,B 0,C 180,E1 -6027.562,E2 -6027.562} C_VEL
LIN {X 0,Y 496,Z 378.808,A -85,B 0,C 180,E1 -6030.1,E2 -6030.1} C_VEL
LIN {X 0,Y 495.877,Z 383.168,A -85,B 0,C 180,E1 -6032.435,E2 -6032.435} C_VEL
LIN {X 0,Y 495.709,Z 389.355,A -85,B 0,C 180,E1 -6035.694,E2 -6035.694} C_VEL
LIN {X 0,Y 495.566,Z 394.09,A -85,B 0,C 180,E1 -6038.151,E2 -6038.151} C_VEL
LIN {X 0,Y 495.472,Z 400.523,A -85,B 0,C 180,E1 -6041.452,E2 -6041.452} C_VEL
LIN {X 0,Y 495.313,Z 407.113,A -85,B 0,C 180,E1 -6044.795,E2 -6044.795} C_VEL
LIN {X 0,Y 495.162,Z 413.907,A -85,B 0,C 180,E1 -6048.193,E2 -6048.193} C_VEL
LIN {X 0,Y 495.119,Z 420.485,A -85,B 0,C 180,E1 -6051.436,E2 -6051.436} C_VEL
LIN {X 0,Y 495.099,Z 420.657,A -85,B 0,C 180,E1 -6051.519,E2 -6051.519} C_VEL
LIN {X 0,Y 496.811,Z 431.31,A -85,B 0,C 180,E1 -6051.905,E2 -6051.905} C_VEL
LIN {X 0,Y 496.65,Z 442.238,A -85,B 0,C 180,E1 -6052.405,E2 -6052.405} C_VEL
LIN {X 0,Y 496.342,Z 452.217,A -85,B 0,C 180,E1 -6053.02,E2 -6053.02} C_VEL
LIN {X 0,Y 496.091,Z 462.091,A -85,B 0,C 180,E1 -6053.81,E2 -6053.81} C_VEL
LIN {X 0,Y 495.891,Z 470.242,A -85,B 0,C 180,E1 -6054.634,E2 -6054.634} C_VEL
LIN {X 0,Y 495.602,Z 478.103,A -85,B 0,C 180,E1 -6055.624,E2 -6055.624} C_VEL
LIN {X 0,Y 495.453,Z 484.656,A -85,B 0,C 180,E1 -6056.665,E2 -6056.665} C_VEL
LIN {X 0,Y 495.263,Z 490.783,A -85,B 0,C 180,E1 -6057.92,E2 -6057.92} C_VEL
LIN {X 0,Y 495.173,Z 494.28,A -85,B 0,C 180,E1 -6058.85,E2 -6058.85} C_VEL
LIN {X 0,Y 495.079,Z 497.526,A -85,B 0,C 180,E1 -6060.011,E2 -6060.011} C_VEL
LIN {X 0,Y 494.986,Z 499.01,A -85,B 0,C 180,E1 -6060.737,E2 -6060.737} C_VEL
LIN {X 0,Y 494.947,Z 500.321,A -85,B 0,C 180,E1 -6061.691,E2 -6061.691} C_VEL
LIN {X 0,Y 494.954,Z 501.026,A -85,B 0,C 180,E1 -6063.096,E2 -6063.096} C_VEL
LIN {X 0,Y 494.983,Z 500.123,A -85,B 0,C 180,E1 -6064.603,E2 -6064.603} C_VEL
LIN {X 0,Y 495.112,Z 497.768,A -85,B 0,C 180,E1 -6065.992,E2 -6065.992} C_VEL
LIN {X 0,Y 495.182,Z 495.155,A -85,B 0,C 180,E1 -6066.978,E2 -6066.978} C_VEL
LIN {X 0,Y 495.25,Z 491.095,A -85,B 0,C 180,E1 -6068.116,E2 -6068.116} C_VEL
LIN {X 0,Y 495.39,Z 486.257,A -85,B 0,C 180,E1 -6069.154,E2 -6069.154} C_VEL
LIN {X 0,Y 495.63,Z 479.243,A -85,B 0,C 180,E1 -6070.323,E2 -6070.323} C_VEL
LIN {X 0,Y 495.823,Z 471.774,A -85,B 0,C 180,E1 -6071.302,E2 -6071.302} C_VEL
LIN {X 0,Y 496.077,Z 463.689,A -85,B 0,C 180,E1 -6072.154,E2 -6072.154} C_VEL
LIN {X 0,Y 496.408,Z 454.199,A -85,B 0,C 180,E1 -6072.945,E2 -6072.945} C_VEL
LIN {X 0,Y 496.687,Z 443.921,A -85,B 0,C 180,E1 -6073.61,E2 -6073.61} C_VEL
LIN {X 0,Y 496.878,Z 433.177,A -85,B 0,C 180,E1 -6074.127,E2 -6074.127} C_VEL
LIN {X 0,Y 496.188,Z 426.359,A -85,B 0,C 180,E1 -6074.394,E2 -6074.394} C_VEL
LIN {X 0,Y 495.161,Z 420.82,A -85,B 0,C 180,E1 -6074.585,E2 -6074.585} C_VEL
LIN {X 0,Y 495.196,Z 414.832,A -85,B 0,C 180,E1 -6077.557,E2 -6077.557} C_VEL
LIN {X 0,Y 495.256,Z 409.364,A -85,B 0,C 180,E1 -6080.314,E2 -6080.314} C_VEL
LIN {X 0,Y 495.367,Z 403.234,A -85,B 0,C 180,E1 -6083.425,E2 -6083.425} C_VEL
LIN {X 0,Y 495.466,Z 399.361,A -85,B 0,C 180,E1 -6085.432,E2 -6085.432} C_VEL
LIN {X 0,Y 495.572,Z 393.684,A -85,B 0,C 180,E1 -6088.351,E2 -6088.351} C_VEL
LIN {X 0,Y 495.722,Z 387.649,A -85,B 0,C 180,E1 -6091.515,E2 -6091.515} C_VEL
LIN {X 0,Y 495.847,Z 383.041,A -85,B 0,C 180,E1 -6093.936,E2 -6093.936} C_VEL
LIN {X 0,Y 495.834,Z 378.726,A -85,B 0,C 180,E1 -6096.285,E2 -6096.285} C_VEL
LIN {X 0,Y 495.755,Z 378.736,A -85,B 0,C 180,E1 -6099.323,E2 -6099.323} C_VEL
LIN {X 0,Y 495.773,Z 378.735,A -85,B 0,C 180,E1 -6101.828,E2 -6101.828} C_VEL
LIN {X 0,Y 495.798,Z 378.731,A -85,B 0,C 180,E1 -6104.548,E2 -6104.548} C_VEL
LIN {X 0,Y 495.854,Z 378.72,A -85,B 0,C 180,E1 -6107.937,E2 -6107.937} C_VEL
LIN {X 0,Y 495.84,Z 378.724,A -85,B 0,C 180,E1 -6111.031,E2 -6111.031} C_VEL
LIN {X 0,Y 495.859,Z 378.72,A -85,B 0,C 180,E1 -6113.49,E2 -6113.49} C_VEL
LIN {X 0,Y 495.849,Z 378.724,A -85,B 0,C 180,E1 -6116.75,E2 -6116.75} C_VEL
LIN {X 0,Y 495.984,Z 378.704,A -85,B 0,C 180,E1 -6119.188,E2 -6119.188} C_VEL
LIN {X 0,Y 495.851,Z 378.719,A -85,B 0,C 180,E1 -6121.625,E2 -6121.625} C_VEL
LIN {X 0,Y 495.848,Z 378.722,A -85,B 0,C 180,E1 -6123.25,E2 -6123.25} C_VEL
LIN {X 0,Y 495.86,Z 378.716,A -85,B 0,C 180,E1 -6126.511,E2 -6126.511} C_VEL
LIN {X 0,Y 495.826,Z 378.722,A -85,B 0,C 180,E1 -6128.97,E2 -6128.97} C_VEL
LIN {X 0,Y 495.831,Z 378.722,A -85,B 0,C 180,E1 -6132.276,E2 -6132.276} C_VEL
LIN {X 0,Y 495.786,Z 378.728,A -85,B 0,C 180,E1 -6135.625,E2 -6135.625} C_VEL
LIN {X 0,Y 495.808,Z 378.725,A -85,B 0,C 180,E1 -6138.257,E2 -6138.257} C_VEL
LIN {X 0,Y 495.744,Z 378.732,A -85,B 0,C 180,E1 -6141.629,E2 -6141.629} C_VEL
LIN {X 0,Y 495.738,Z 378.733,A -85,B 0,C 180,E1 -6144.276,E2 -6144.276} C_VEL
LIN {X 0,Y 495.8,Z 378.726,A -85,B 0,C 180,E1 -6146.975,E2 -6146.975} C_VEL
LIN {X 0,Y 495.757,Z 378.733,A -85,B 0,C 180,E1 -6150.151,E2 -6150.151} C_VEL
LIN {X 0,Y 495.775,Z 378.729,A -85,B 0,C 180,E1 -6153.247,E2 -6153.247} C_VEL
LIN {X 0,Y 495.711,Z 378.738,A -85,B 0,C 180,E1 -6156.092,E2 -6156.092} C_VEL
LIN {X 0,Y 495.761,Z 378.731,A -85,B 0,C 180,E1 -6158.773,E2 -6158.773} C_VEL
LIN {X 0,Y 495.767,Z 378.732,A -85,B 0,C 180,E1 -6161.78,E2 -6161.78} C_VEL
LIN {X 0,Y 495.735,Z 378.734,A -85,B 0,C 180,E1 -6165.142,E2 -6165.142} C_VEL
LIN {X 0,Y 495.766,Z 378.731,A -85,B 0,C 180,E1 -6168.224,E2 -6168.224} C_VEL
LIN {X 0,Y 495.767,Z 378.733,A -85,B 0,C 180,E1 -6171.232,E2 -6171.232} C_VEL
LIN {X 0,Y 495.748,Z 378.735,A -85,B 0,C 180,E1 -6174.466,E2 -6174.466} C_VEL
LIN {X 0,Y 495.795,Z 378.779,A -85,B 0,C 180,E1 -6176.32,E2 -6176.32} C_VEL
LIN {X 0,Y 497.352,Z 386.894,A -85,B 0,C 180,E1 -6178.954,E2 -6178.954} C_VEL
LIN {X 0,Y 497.528,Z 391.599,A -85,B 0,C 180,E1 -6180.372,E2 -6180.372} C_VEL
LIN {X 0,Y 497.041,Z 401.179,A -85,B 0,C 180,E1 -6183.101,E2 -6183.101} C_VEL
LIN {X 0,Y 496.558,Z 412.502,A -85,B 0,C 180,E1 -6186.213,E2 -6186.213} C_VEL
LIN {X 0,Y 496.125,Z 423.992,A -85,B 0,C 180,E1 -6189.261,E2 -6189.261} C_VEL
LIN {X 0,Y 495.762,Z 437.345,A -85,B 0,C 180,E1 -6192.683,E2 -6192.683} C_VEL
LIN {X 0,Y 495.55,Z 449.047,A -85,B 0,C 180,E1 -6195.593,E2 -6195.593} C_VEL
LIN {X 0,Y 497.325,Z 462.069,A -85,B 0,C 180,E1 -6195.932,E2 -6195.932} C_VEL
LIN {X 0,Y 497.507,Z 467.417,A -85,B 0,C 180,E1 -6196.107,E2 -6196.107} C_VEL
LIN {X 0,Y 497.113,Z 480.006,A -85,B 0,C 180,E1 -6196.617,E2 -6196.617} C_VEL
LIN {X 0,Y 496.784,Z 491.199,A -85,B 0,C 180,E1 -6197.232,E2 -6197.232} C_VEL
LIN {X 0,Y 496.46,Z 502.824,A -85,B 0,C 180,E1 -6198.054,E2 -6198.054} C_VEL
LIN {X 0,Y 496.098,Z 513.28,A -85,B 0,C 180,E1 -6198.976,E2 -6198.976} C_VEL
LIN {X 0,Y 495.761,Z 522.657,A -85,B 0,C 180,E1 -6200.002,E2 -6200.002} C_VEL
LIN {X 0,Y 495.484,Z 531.734,A -85,B 0,C 180,E1 -6201.231,E2 -6201.231} C_VEL
LIN {X 0,Y 495.284,Z 539.042,A -85,B 0,C 180,E1 -6202.46,E2 -6202.46} C_VEL
LIN {X 0,Y 495.134,Z 545.127,A -85,B 0,C 180,E1 -6203.749,E2 -6203.749} C_VEL
LIN {X 0,Y 495.038,Z 550.09,A -85,B 0,C 180,E1 -6205.115,E2 -6205.115} C_VEL
LIN {X 0,Y 495.056,Z 552.419,A -85,B 0,C 180,E1 -6205.932,E2 -6205.932} C_VEL
LIN {X 0,Y 495.044,Z 554.308,A -85,B 0,C 180,E1 -6206.746,E2 -6206.746} C_VEL
LIN {X 0,Y 495.054,Z 555.724,A -85,B 0,C 180,E1 -6207.561,E2 -6207.561} C_VEL
LIN {X 0,Y 494.911,Z 557.339,A -85,B 0,C 180,E1 -6209.188,E2 -6209.188} C_VEL
LIN {X 0,Y 494.899,Z 557.559,A -85,B 0,C 180,E1 -6210.002,E2 -6210.002} C_VEL
LIN {X 0,Y 494.963,Z 556.732,A -85,B 0,C 180,E1 -6211.629,E2 -6211.629} C_VEL
LIN {X 0,Y 495.054,Z 555.734,A -85,B 0,C 180,E1 -6212.443,E2 -6212.443} C_VEL
LIN {X 0,Y 495.045,Z 554.322,A -85,B 0,C 180,E1 -6213.257,E2 -6213.257} C_VEL
LIN {X 0,Y 495.019,Z 551.359,A -85,B 0,C 180,E1 -6214.48,E2 -6214.48} C_VEL
LIN {X 0,Y 495.155,Z 547.351,A -85,B 0,C 180,E1 -6215.704,E2 -6215.704} C_VEL
LIN {X 0,Y 495.259,Z 541.157,A -85,B 0,C 180,E1 -6217.134,E2 -6217.134} C_VEL
LIN {X 0,Y 495.436,Z 534.4,A -85,B 0,C 180,E1 -6218.362,E2 -6218.362} C_VEL
LIN {X 0,Y 495.679,Z 526.005,A -85,B 0,C 180,E1 -6219.592,E2 -6219.592} C_VEL
LIN {X 0,Y 495.992,Z 517.346,A -85,B 0,C 180,E1 -6220.616,E2 -6220.616} C_VEL
LIN {X 0,Y 496.375,Z 506.662,A -85,B 0,C 180,E1 -6221.641,E2 -6221.641} C_VEL
LIN {X 0,Y 496.637,Z 496.054,A -85,B 0,C 180,E1 -6222.463,E2 -6222.463} C_VEL
LIN {X 0,Y 497.04,Z 484.191,A -85,B 0,C 180,E1 -6223.181,E2 -6223.181} C_VEL
LIN {X 0,Y 497.386,Z 471.836,A -85,B 0,C 180,E1 -6223.744,E2 -6223.744} C_VEL
LIN {X 0,Y 497.457,Z 462.79,A -85,B 0,C 180,E1 -6224.055,E2 -6224.055} C_VEL
LIN {X 0,Y 495.713,Z 450.4,A -85,B 0,C 180,E1 -6224.39,E2 -6224.39} C_VEL
LIN {X 0,Y 495.531,Z 448.964,A -85,B 0,C 180,E1 -6224.425,E2 -6224.425} C_VEL
LIN {X 0,Y 495.772,Z 437.55,A -85,B 0,C 180,E1 -6227.321,E2 -6227.321} C_VEL
LIN {X 0,Y 496.088,Z 425.891,A -85,B 0,C 180,E1 -6230.311,E2 -6230.311} C_VEL
LIN {X 0,Y 496.503,Z 414.312,A -85,B 0,C 180,E1 -6233.351,E2 -6233.351} C_VEL
LIN {X 0,Y 496.965,Z 402.875,A -85,B 0,C 180,E1 -6236.455,E2 -6236.455} C_VEL
LIN {X 0,Y 497.488,Z 393.089,A -85,B 0,C 180,E1 -6239.181,E2 -6239.181} C_VEL
LIN {X 0,Y 497.502,Z 388.295,A -85,B 0,C 180,E1 -6240.569,E2 -6240.569} C_VEL
LIN {X 0,Y 496.194,Z 380.745,A -85,B 0,C 180,E1 -6242.909,E2 -6242.909} C_VEL
LIN {X 0,Y 495.802,Z 378.728,A -85,B 0,C 180,E1 -6243.562,E2 -6243.562} C_VEL
LIN {X 0,Y 495.723,Z 378.739,A -85,B 0,C 180,E1 -6246.546,E2 -6246.546} C_VEL
LIN {X 0,Y 495.75,Z 378.734,A -85,B 0,C 180,E1 -6249.64,E2 -6249.64} C_VEL
LIN {X 0,Y 495.695,Z 378.738,A -85,B 0,C 180,E1 -6252.888,E2 -6252.888} C_VEL
LIN {X 0,Y 495.728,Z 378.73,A -85,B 0,C 180,E1 -6255.998,E2 -6255.998} C_VEL
LIN {X 0,Y 495.737,Z 378.733,A -85,B 0,C 180,E1 -6259.297,E2 -6259.297} C_VEL
LIN {X 0,Y 495.753,Z 378.728,A -85,B 0,C 180,E1 -6261.408,E2 -6261.408} C_VEL
LIN {X 0,Y 495.753,Z 378.735,A -85,B 0,C 180,E1 -6264.462,E2 -6264.462} C_VEL
LIN {X 0,Y 495.757,Z 378.73,A -85,B 0,C 180,E1 -6267.405,E2 -6267.405} C_VEL
LIN {X 0,Y 495.762,Z 378.729,A -85,B 0,C 180,E1 -6270.253,E2 -6270.253} C_VEL
LIN {X 0,Y 495.725,Z 378.738,A -85,B 0,C 180,E1 -6273.275,E2 -6273.275} C_VEL
LIN {X 0,Y 495.707,Z 378.735,A -85,B 0,C 180,E1 -6275.722,E2 -6275.722} C_VEL
LIN {X 0,Y 495.746,Z 378.734,A -85,B 0,C 180,E1 -6278.371,E2 -6278.371} C_VEL
LIN {X 0,Y 495.788,Z 378.727,A -85,B 0,C 180,E1 -6280.971,E2 -6280.971} C_VEL
LIN {X 0,Y 495.782,Z 378.728,A -85,B 0,C 180,E1 -6283.53,E2 -6283.53} C_VEL
LIN {X 0,Y 495.795,Z 378.73,A -85,B 0,C 180,E1 -6286.055,E2 -6286.055} C_VEL
LIN {X 0,Y 495.852,Z 378.718,A -85,B 0,C 180,E1 -6288.555,E2 -6288.555} C_VEL
LIN {X 0,Y 495.813,Z 378.724,A -85,B 0,C 180,E1 -6291.851,E2 -6291.851} C_VEL
LIN {X 0,Y 495.862,Z 378.719,A -85,B 0,C 180,E1 -6294.306,E2 -6294.306} C_VEL
LIN {X 0,Y 495.538,Z 378.878,A -85,B 0,C 180,E1 -6297.053,E2 -6297.053} C_VEL
LIN {X 0,Y 495.721,Z 386.152,A -85,B 0,C 180,E1 -6300,E2 -6300} C_VEL
LIN {X 0,Y 495.421,Z 392.081,A -85,B 0,C 180,E1 -6302.439,E2 -6302.439} C_VEL
LIN {X 0,Y 495.503,Z 397.847,A -85,B 0,C 180,E1 -6304.882,E2 -6304.882} C_VEL
LIN {X 0,Y 495.438,Z 403.47,A -85,B 0,C 180,E1 -6307.335,E2 -6307.335} C_VEL
LIN {X 0,Y 495.366,Z 411.139,A -85,B 0,C 180,E1 -6310.628,E2 -6310.628} C_VEL
LIN {X 0,Y 495.258,Z 416.793,A -85,B 0,C 180,E1 -6313.123,E2 -6313.123} C_VEL
LIN {X 0,Y 495.194,Z 422.472,A -85,B 0,C 180,E1 -6315.643,E2 -6315.643} C_VEL
LIN {X 0,Y 495.159,Z 424.551,A -85,B 0,C 180,E1 -6316.57,E2 -6316.57} C_VEL
LIN {X 0,Y 497.669,Z 438.099,A -85,B 0,C 180,E1 -6317.013,E2 -6317.013} C_VEL
LIN {X 0,Y 497.449,Z 450.969,A -85,B 0,C 180,E1 -6317.524,E2 -6317.524} C_VEL
LIN {X 0,Y 497.023,Z 463.291,A -85,B 0,C 180,E1 -6318.19,E2 -6318.19} C_VEL
LIN {X 0,Y 496.689,Z 474.747,A -85,B 0,C 180,E1 -6318.992,E2 -6318.992} C_VEL
LIN {X 0,Y 496.311,Z 485.789,A -85,B 0,C 180,E1 -6319.975,E2 -6319.975} C_VEL
LIN {X 0,Y 495.967,Z 494.637,A -85,B 0,C 180,E1 -6320.943,E2 -6320.943} C_VEL
LIN {X 0,Y 495.686,Z 503.073,A -85,B 0,C 180,E1 -6322.069,E2 -6322.069} C_VEL
LIN {X 0,Y 495.446,Z 511.037,A -85,B 0,C 180,E1 -6323.402,E2 -6323.402} C_VEL
LIN {X 0,Y 495.179,Z 517.295,A -85,B 0,C 180,E1 -6324.721,E2 -6324.721} C_VEL
LIN {X 0,Y 495.096,Z 522.305,A -85,B 0,C 180,E1 -6326.107,E2 -6326.107} C_VEL
LIN {X 0,Y 494.986,Z 525.915,A -85,B 0,C 180,E1 -6327.48,E2 -6327.48} C_VEL
LIN {X 0,Y 494.927,Z 528.328,A -85,B 0,C 180,E1 -6328.868,E2 -6328.868} C_VEL
LIN {X 0,Y 494.929,Z 529.406,A -85,B 0,C 180,E1 -6329.979,E2 -6329.979} C_VEL
LIN {X 0,Y 494.892,Z 529.668,A -85,B 0,C 180,E1 -6331.562,E2 -6331.562} C_VEL
LIN {X 0,Y 494.919,Z 528.49,A -85,B 0,C 180,E1 -6333.088,E2 -6333.088} C_VEL
LIN {X 0,Y 495.003,Z 525.893,A -85,B 0,C 180,E1 -6334.605,E2 -6334.605} C_VEL
LIN {X 0,Y 495.08,Z 522.252,A -85,B 0,C 180,E1 -6335.985,E2 -6335.985} C_VEL
LIN {X 0,Y 495.238,Z 517.219,A -85,B 0,C 180,E1 -6337.372,E2 -6337.372} C_VEL
LIN {X 0,Y 495.385,Z 510.849,A -85,B 0,C 180,E1 -6338.712,E2 -6338.712} C_VEL
LIN {X 0,Y 495.647,Z 502.941,A -85,B 0,C 180,E1 -6340.03,E2 -6340.03} C_VEL
LIN {X 0,Y 495.945,Z 494.401,A -85,B 0,C 180,E1 -6341.165,E2 -6341.165} C_VEL
LIN {X 0,Y 496.307,Z 484.139,A -85,B 0,C 180,E1 -6342.27,E2 -6342.27} C_VEL
LIN {X 0,Y 496.695,Z 473.411,A -85,B 0,C 180,E1 -6343.195,E2 -6343.195} C_VEL
LIN {X 0,Y 497.067,Z 461.696,A -85,B 0,C 180,E1 -6343.993,E2 -6343.993} C_VEL
LIN {X 0,Y 497.43,Z 450.455,A -85,B 0,C 180,E1 -6344.589,E2 -6344.589} C_VEL
LIN {X 0,Y 497.641,Z 438.081,A -85,B 0,C 180,E1 -6345.078,E2 -6345.078} C_VEL
LIN {X 0,Y 495.427,Z 425.786,A -85,B 0,C 180,E1 -6345.476,E2 -6345.476} C_VEL
LIN {X 0,Y 495.191,Z 424.302,A -85,B 0,C 180,E1 -6345.539,E2 -6345.539} C_VEL
LIN {X 0,Y 495.25,Z 417.559,A -85,B 0,C 180,E1 -6348.579,E2 -6348.579} C_VEL
LIN {X 0,Y 494.614,Z 416.149,A -85,B 0,C 180,E1 -6349.238,E2 -6349.238} C_VEL
LIN {X 0,Y 491.785,Z 414.034,A -85,B 0,C 180,E1 -6350.314,E2 -6350.314} C_VEL
LIN {X 0,Y 489.375,Z 412.357,A -85,B 0,C 180,E1 -6351.182,E2 -6351.182} C_VEL
LIN {X 0,Y 488.335,Z 410.984,A -85,B 0,C 180,E1 -6351.85,E2 -6351.85} C_VEL
LIN {X 0,Y 488.248,Z 410.497,A -85,B 0,C 180,E1 -6352.075,E2 -6352.075} C_VEL
LIN {X 0,Y 488.389,Z 403.806,A -85,B 0,C 180,E1 -6355.108,E2 -6355.108} C_VEL
LIN {X 0,Y 488.467,Z 397.204,A -85,B 0,C 180,E1 -6358.09,E2 -6358.09} C_VEL
LIN {X 0,Y 488.503,Z 391.417,A -85,B 0,C 180,E1 -6360.714,E2 -6360.714} C_VEL
LIN {X 0,Y 488.569,Z 385.2,A -85,B 0,C 180,E1 -6363.516,E2 -6363.516} C_VEL
LIN {X 0,Y 488.755,Z 379.607,A -85,B 0,C 180,E1 -6366.031,E2 -6366.031} C_VEL
LIN {X 0,Y 488.749,Z 379.606,A -85,B 0,C 180,E1 -6369.174,E2 -6369.174} C_VEL
LIN {X 0,Y 488.749,Z 379.605,A -85,B 0,C 180,E1 -6371.631,E2 -6371.631} C_VEL
LIN {X 0,Y 488.764,Z 379.605,A -85,B 0,C 180,E1 -6374.998,E2 -6374.998} C_VEL
LIN {X 0,Y 488.806,Z 379.601,A -85,B 0,C 180,E1 -6378.386,E2 -6378.386} C_VEL
LIN {X 0,Y 488.817,Z 379.597,A -85,B 0,C 180,E1 -6381.732,E2 -6381.732} C_VEL
LIN {X 0,Y 488.802,Z 379.6,A -85,B 0,C 180,E1 -6385.049,E2 -6385.049} C_VEL
LIN {X 0,Y 488.943,Z 379.582,A -85,B 0,C 180,E1 -6387.527,E2 -6387.527} C_VEL
LIN {X 0,Y 488.958,Z 379.619,A -85,B 0,C 180,E1 -6389.998,E2 -6389.998} C_VEL
LIN {X 0,Y 488.827,Z 384.182,A -85,B 0,C 180,E1 -6392.47,E2 -6392.47} C_VEL
LIN {X 0,Y 488.67,Z 390.409,A -85,B 0,C 180,E1 -6395.776,E2 -6395.776} C_VEL
LIN {X 0,Y 488.521,Z 395.158,A -85,B 0,C 180,E1 -6398.269,E2 -6398.269} C_VEL
LIN {X 0,Y 488.431,Z 402.192,A -85,B 0,C 180,E1 -6401.918,E2 -6401.918} C_VEL
LIN {X 0,Y 488.221,Z 408.863,A -85,B 0,C 180,E1 -6405.32,E2 -6405.32} C_VEL
LIN {X 0,Y 488.096,Z 415.089,A -85,B 0,C 180,E1 -6408.466,E2 -6408.466} C_VEL
LIN {X 0,Y 488.037,Z 420.816,A -85,B 0,C 180,E1 -6411.32,E2 -6411.32} C_VEL
LIN {X 0,Y 489.952,Z 432.883,A -85,B 0,C 180,E1 -6411.784,E2 -6411.784} C_VEL
LIN {X 0,Y 489.695,Z 443.597,A -85,B 0,C 180,E1 -6412.296,E2 -6412.296} C_VEL
LIN {X 0,Y 489.369,Z 453.452,A -85,B 0,C 180,E1 -6412.93,E2 -6412.93} C_VEL
LIN {X 0,Y 489.085,Z 463.063,A -85,B 0,C 180,E1 -6413.723,E2 -6413.723} C_VEL
LIN {X 0,Y 488.848,Z 471.748,A -85,B 0,C 180,E1 -6414.638,E2 -6414.638} C_VEL
LIN {X 0,Y 488.573,Z 478.849,A -85,B 0,C 180,E1 -6415.563,E2 -6415.563} C_VEL
LIN {X 0,Y 488.337,Z 486.501,A -85,B 0,C 180,E1 -6416.839,E2 -6416.839} C_VEL
LIN {X 0,Y 488.214,Z 491.375,A -85,B 0,C 180,E1 -6417.892,E2 -6417.892} C_VEL
LIN {X 0,Y 488.117,Z 495.016,A -85,B 0,C 180,E1 -6418.896,E2 -6418.896} C_VEL
LIN {X 0,Y 487.964,Z 498.587,A -85,B 0,C 180,E1 -6420.268,E2 -6420.268} C_VEL
LIN {X 0,Y 487.854,Z 500.845,A -85,B 0,C 180,E1 -6421.794,E2 -6421.794} C_VEL
LIN {X 0,Y 487.859,Z 501.39,A -85,B 0,C 180,E1 -6423.329,E2 -6423.329} C_VEL
LIN {X 0,Y 487.871,Z 500.982,A -85,B 0,C 180,E1 -6424.178,E2 -6424.178} C_VEL
LIN {X 0,Y 487.939,Z 499.814,A -85,B 0,C 180,E1 -6425.176,E2 -6425.176} C_VEL
LIN {X 0,Y 488.077,Z 496.578,A -85,B 0,C 180,E1 -6426.696,E2 -6426.696} C_VEL
LIN {X 0,Y 488.158,Z 492.601,A -85,B 0,C 180,E1 -6427.912,E2 -6427.912} C_VEL
LIN {X 0,Y 488.326,Z 487.895,A -85,B 0,C 180,E1 -6428.998,E2 -6428.998} C_VEL
LIN {X 0,Y 488.505,Z 482.025,A -85,B 0,C 180,E1 -6430.066,E2 -6430.066} C_VEL
LIN {X 0,Y 488.769,Z 474.573,A -85,B 0,C 180,E1 -6431.132,E2 -6431.132} C_VEL
LIN {X 0,Y 489.036,Z 465.805,A -85,B 0,C 180,E1 -6432.125,E2 -6432.125} C_VEL
LIN {X 0,Y 489.401,Z 455.984,A -85,B 0,C 180,E1 -6432.994,E2 -6432.994} C_VEL
LIN {X 0,Y 489.694,Z 446.218,A -85,B 0,C 180,E1 -6433.662,E2 -6433.662} C_VEL
LIN {X 0,Y 489.956,Z 435.428,A -85,B 0,C 180,E1 -6434.222,E2 -6434.222} C_VEL
LIN {X 0,Y 489.595,Z 429.426,A -85,B 0,C 180,E1 -6434.471,E2 -6434.471} C_VEL
LIN {X 0,Y 488.083,Z 421.05,A -85,B 0,C 180,E1 -6434.79,E2 -6434.79} C_VEL
LIN {X 0,Y 488.138,Z 414.693,A -85,B 0,C 180,E1 -6437.973,E2 -6437.973} C_VEL
LIN {X 0,Y 488.198,Z 408.732,A -85,B 0,C 180,E1 -6441.016,E2 -6441.016} C_VEL
LIN {X 0,Y 488.336,Z 403.265,A -85,B 0,C 180,E1 -6443.839,E2 -6443.839} C_VEL
LIN {X 0,Y 488.452,Z 397.452,A -85,B 0,C 180,E1 -6446.856,E2 -6446.856} C_VEL
LIN {X 0,Y 488.581,Z 391.887,A -85,B 0,C 180,E1 -6449.771,E2 -6449.771} C_VEL
LIN {X 0,Y 488.773,Z 385.705,A -85,B 0,C 180,E1 -6453.054,E2 -6453.054} C_VEL
LIN {X 0,Y 488.862,Z 381.401,A -85,B 0,C 180,E1 -6455.361,E2 -6455.361} C_VEL
LIN {X 0,Y 488.783,Z 379.605,A -85,B 0,C 180,E1 -6456.37,E2 -6456.37} C_VEL
LIN {X 0,Y 488.706,Z 379.612,A -85,B 0,C 180,E1 -6459.81,E2 -6459.81} C_VEL
LIN {X 0,Y 488.711,Z 379.613,A -85,B 0,C 180,E1 -6462.423,E2 -6462.423} C_VEL
LIN {X 0,Y 488.741,Z 379.608,A -85,B 0,C 180,E1 -6464.999,E2 -6464.999} C_VEL
LIN {X 0,Y 488.813,Z 379.599,A -85,B 0,C 180,E1 -6468.388,E2 -6468.388} C_VEL
LIN {X 0,Y 488.801,Z 379.598,A -85,B 0,C 180,E1 -6471.734,E2 -6471.734} C_VEL
LIN {X 0,Y 488.851,Z 379.594,A -85,B 0,C 180,E1 -6474.224,E2 -6474.224} C_VEL
LIN {X 0,Y 488.946,Z 379.581,A -85,B 0,C 180,E1 -6477.529,E2 -6477.529} C_VEL
LIN {X 0,Y 488.943,Z 379.581,A -85,B 0,C 180,E1 -6480,E2 -6480} C_VEL
LIN {X 0,Y 488.946,Z 379.58,A -85,B 0,C 180,E1 -6482.472,E2 -6482.472} C_VEL
LIN {X 0,Y 488.852,Z 379.594,A -85,B 0,C 180,E1 -6485.776,E2 -6485.776} C_VEL
LIN {X 0,Y 488.796,Z 379.6,A -85,B 0,C 180,E1 -6488.267,E2 -6488.267} C_VEL
LIN {X 0,Y 488.814,Z 379.597,A -85,B 0,C 180,E1 -6491.613,E2 -6491.613} C_VEL
LIN {X 0,Y 488.743,Z 379.606,A -85,B 0,C 180,E1 -6495.001,E2 -6495.001} C_VEL
LIN {X 0,Y 488.744,Z 379.603,A -85,B 0,C 180,E1 -6498.443,E2 -6498.443} C_VEL
LIN {X 0,Y 488.72,Z 379.607,A -85,B 0,C 180,E1 -6501.07,E2 -6501.07} C_VEL
LIN {X 0,Y 488.682,Z 379.612,A -85,B 0,C 180,E1 -6503.746,E2 -6503.746} C_VEL
LIN {X 0,Y 488.778,Z 379.6,A -85,B 0,C 180,E1 -6506.947,E2 -6506.947} C_VEL
LIN {X 0,Y 488.699,Z 379.611,A -85,B 0,C 180,E1 -6510.367,E2 -6510.367} C_VEL
LIN {X 0,Y 488.717,Z 379.608,A -85,B 0,C 180,E1 -6513.486,E2 -6513.486} C_VEL
LIN {X 0,Y 488.671,Z 379.615,A -85,B 0,C 180,E1 -6516.358,E2 -6516.358} C_VEL
LIN {X 0,Y 488.732,Z 379.609,A -85,B 0,C 180,E1 -6519.252,E2 -6519.252} C_VEL
LIN {X 0,Y 488.717,Z 379.61,A -85,B 0,C 180,E1 -6522.523,E2 -6522.523} C_VEL
LIN {X 0,Y 488.697,Z 379.61,A -85,B 0,C 180,E1 -6525.201,E2 -6525.201} C_VEL
LIN {X 0,Y 488.722,Z 379.611,A -85,B 0,C 180,E1 -6527.481,E2 -6527.481} C_VEL
LIN {X 0,Y 488.737,Z 379.607,A -85,B 0,C 180,E1 -6530.753,E2 -6530.753} C_VEL
LIN {X 0,Y 488.675,Z 379.617,A -85,B 0,C 180,E1 -6533.871,E2 -6533.871} C_VEL
LIN {X 0,Y 488.757,Z 379.776,A -85,B 0,C 180,E1 -6536.061,E2 -6536.061} C_VEL
LIN {X 0,Y 490.443,Z 388.473,A -85,B 0,C 180,E1 -6538.947,E2 -6538.947} C_VEL
LIN {X 0,Y 490.557,Z 393.164,A -85,B 0,C 180,E1 -6540.382,E2 -6540.382} C_VEL
LIN {X 0,Y 490.02,Z 402.804,A -85,B 0,C 180,E1 -6543.178,E2 -6543.178} C_VEL
LIN {X 0,Y 489.529,Z 414.035,A -85,B 0,C 180,E1 -6546.3,E2 -6546.3} C_VEL
LIN {X 0,Y 489.052,Z 425.646,A -85,B 0,C 180,E1 -6549.443,E2 -6549.443} C_VEL
LIN {X 0,Y 488.693,Z 438.742,A -85,B 0,C 180,E1 -6552.856,E2 -6552.856} C_VEL
LIN {X 0,Y 488.477,Z 448.67,A -85,B 0,C 180,E1 -6555.393,E2 -6555.393} C_VEL
LIN {X 0,Y 490.38,Z 462.902,A -85,B 0,C 180,E1 -6555.782,E2 -6555.782} C_VEL
LIN {X 0,Y 490.462,Z 470.842,A -85,B 0,C 180,E1 -6556.062,E2 -6556.062} C_VEL
LIN {X 0,Y 490.075,Z 483.355,A -85,B 0,C 180,E1 -6556.632,E2 -6556.632} C_VEL
LIN {X 0,Y 489.654,Z 494.749,A -85,B 0,C 180,E1 -6557.318,E2 -6557.318} C_VEL
LIN {X 0,Y 489.3,Z 506.039,A -85,B 0,C 180,E1 -6558.193,E2 -6558.193} C_VEL
LIN {X 0,Y 488.96,Z 516.759,A -85,B 0,C 180,E1 -6559.233,E2 -6559.233} C_VEL
LIN {X 0,Y 488.602,Z 525.459,A -85,B 0,C 180,E1 -6560.272,E2 -6560.272} C_VEL
LIN {X 0,Y 488.36,Z 533.891,A -85,B 0,C 180,E1 -6561.52,E2 -6561.52} C_VEL
LIN {X 0,Y 488.181,Z 540.675,A -85,B 0,C 180,E1 -6562.765,E2 -6562.765} C_VEL
LIN {X 0,Y 488.048,Z 546.889,A -85,B 0,C 180,E1 -6564.217,E2 -6564.217} C_VEL
LIN {X 0,Y 487.929,Z 550.916,A -85,B 0,C 180,E1 -6565.458,E2 -6565.458} C_VEL
LIN {X 0,Y 487.968,Z 553.896,A -85,B 0,C 180,E1 -6566.699,E2 -6566.699} C_VEL
LIN {X 0,Y 487.959,Z 555.314,A -85,B 0,C 180,E1 -6567.525,E2 -6567.525} C_VEL
LIN {X 0,Y 487.834,Z 556.934,A -85,B 0,C 180,E1 -6569.176,E2 -6569.176} C_VEL
LIN {X 0,Y 487.82,Z 557.155,A -85,B 0,C 180,E1 -6570.002,E2 -6570.002} C_VEL
LIN {X 0,Y 487.893,Z 556.33,A -85,B 0,C 180,E1 -6571.653,E2 -6571.653} C_VEL
LIN {X 0,Y 487.96,Z 555.33,A -85,B 0,C 180,E1 -6572.478,E2 -6572.478} C_VEL
LIN {X 0,Y 487.969,Z 553.917,A -85,B 0,C 180,E1 -6573.304,E2 -6573.304} C_VEL
LIN {X 0,Y 487.93,Z 550.951,A -85,B 0,C 180,E1 -6574.545,E2 -6574.545} C_VEL
LIN {X 0,Y 488.051,Z 546.937,A -85,B 0,C 180,E1 -6575.787,E2 -6575.787} C_VEL
LIN {X 0,Y 488.185,Z 540.735,A -85,B 0,C 180,E1 -6577.238,E2 -6577.238} C_VEL
LIN {X 0,Y 488.366,Z 533.967,A -85,B 0,C 180,E1 -6578.484,E2 -6578.484} C_VEL
LIN {X 0,Y 488.606,Z 525.552,A -85,B 0,C 180,E1 -6579.732,E2 -6579.732} C_VEL
LIN {X 0,Y 488.961,Z 516.869,A -85,B 0,C 180,E1 -6580.771,E2 -6580.771} C_VEL
LIN {X 0,Y 489.355,Z 506.168,A -85,B 0,C 180,E1 -6581.81,E2 -6581.81} C_VEL
LIN {X 0,Y 489.656,Z 495.778,A -85,B 0,C 180,E1 -6582.624,E2 -6582.624} C_VEL
LIN {X 0,Y 490.056,Z 483.55,A -85,B 0,C 180,E1 -6583.372,E2 -6583.372} C_VEL
LIN {X 0,Y 490.449,Z 471.088,A -85,B 0,C 180,E1 -6583.942,E2 -6583.942} C_VEL
LIN {X 0,Y 490.442,Z 463.219,A -85,B 0,C 180,E1 -6584.22,E2 -6584.22} C_VEL
LIN {X 0,Y 488.664,Z 450.313,A -85,B 0,C 180,E1 -6584.579,E2 -6584.579} C_VEL
LIN {X 0,Y 488.482,Z 448.711,A -85,B 0,C 180,E1 -6584.638,E2 -6584.638} C_VEL
LIN {X 0,Y 488.784,Z 435.726,A -85,B 0,C 180,E1 -6587.983,E2 -6587.983} C_VEL
LIN {X 0,Y 489.155,Z 424.02,A -85,B 0,C 180,E1 -6591.052,E2 -6591.052} C_VEL
LIN {X 0,Y 489.619,Z 412.553,A -85,B 0,C 180,E1 -6594.149,E2 -6594.149} C_VEL
LIN {X 0,Y 490.137,Z 401.129,A -85,B 0,C 180,E1 -6597.314,E2 -6597.314} C_VEL
LIN {X 0,Y 490.624,Z 391.471,A -85,B 0,C 180,E1 -6600.091,E2 -6600.091} C_VEL
LIN {X 0,Y 490.082,Z 386.64,A -85,B 0,C 180,E1 -6601.564,E2 -6601.564} C_VEL
LIN {X 0,Y 488.756,Z 379.607,A -85,B 0,C 180,E1 -6603.853,E2 -6603.853} C_VEL
LIN {X 0,Y 488.677,Z 379.613,A -85,B 0,C 180,E1 -6607.16,E2 -6607.16} C_VEL
LIN {X 0,Y 488.7,Z 379.611,A -85,B 0,C 180,E1 -6610.342,E2 -6610.342} C_VEL
LIN {X 0,Y 488.67,Z 379.617,A -85,B 0,C 180,E1 -6613.658,E2 -6613.658} C_VEL
LIN {X 0,Y 488.68,Z 379.607,A -85,B 0,C 180,E1 -6616.344,E2 -6616.344} C_VEL
LIN {X 0,Y 488.709,Z 379.606,A -85,B 0,C 180,E1 -6619.674,E2 -6619.674} C_VEL
LIN {X 0,Y 488.685,Z 379.613,A -85,B 0,C 180,E1 -6622.841,E2 -6622.841} C_VEL
LIN {X 0,Y 488.726,Z 379.609,A -85,B 0,C 180,E1 -6625.887,E2 -6625.887} C_VEL
LIN {X 0,Y 488.694,Z 379.608,A -85,B 0,C 180,E1 -6628.82,E2 -6628.82} C_VEL
LIN {X 0,Y 488.697,Z 379.613,A -85,B 0,C 180,E1 -6631.668,E2 -6631.668} C_VEL
LIN {X 0,Y 488.695,Z 379.613,A -85,B 0,C 180,E1 -6634.961,E2 -6634.961} C_VEL
LIN {X 0,Y 488.702,Z 379.609,A -85,B 0,C 180,E1 -6638.043,E2 -6638.043} C_VEL
LIN {X 0,Y 488.748,Z 379.607,A -85,B 0,C 180,E1 -6640.687,E2 -6640.687} C_VEL
LIN {X 0,Y 488.768,Z 379.606,A -85,B 0,C 180,E1 -6644.145,E2 -6644.145} C_VEL
LIN {X 0,Y 488.744,Z 379.609,A -85,B 0,C 180,E1 -6647.543,E2 -6647.543} C_VEL
LIN {X 0,Y 488.745,Z 379.604,A -85,B 0,C 180,E1 -6650.063,E2 -6650.063} C_VEL
LIN {X 0,Y 488.823,Z 379.598,A -85,B 0,C 180,E1 -6652.769,E2 -6652.769} C_VEL
LIN {X 0,Y 488.793,Z 379.602,A -85,B 0,C 180,E1 -6655.051,E2 -6655.051} C_VEL
LIN {X 0,Y 488.52,Z 379.734,A -85,B 0,C 180,E1 -6657.01,E2 -6657.01} C_VEL
LIN {X 0,Y 488.683,Z 387.074,A -85,B 0,C 180,E1 -6660,E2 -6660} C_VEL
LIN {X 0,Y 488.369,Z 393.036,A -85,B 0,C 180,E1 -6662.474,E2 -6662.474} C_VEL
LIN {X 0,Y 488.448,Z 398.821,A -85,B 0,C 180,E1 -6664.952,E2 -6664.952} C_VEL
LIN {X 0,Y 488.393,Z 404.544,A -85,B 0,C 180,E1 -6667.441,E2 -6667.441} C_VEL
LIN {X 0,Y 488.303,Z 412.219,A -85,B 0,C 180,E1 -6670.784,E2 -6670.784} C_VEL
LIN {X 0,Y 488.169,Z 417.911,A -85,B 0,C 180,E1 -6673.317,E2 -6673.317} C_VEL
LIN {X 0,Y 488.113,Z 423.644,A -85,B 0,C 180,E1 -6675.876,E2 -6675.876} C_VEL
LIN {X 0,Y 488.088,Z 424.738,A -85,B 0,C 180,E1 -6676.36,E2 -6676.36} C_VEL
LIN {X 0,Y 490.55,Z 437.539,A -85,B 0,C 180,E1 -6676.784,E2 -6676.784} C_VEL
LIN {X 0,Y 490.748,Z 442.422,A -85,B 0,C 180,E1 -6676.965,E2 -6676.965} C_VEL
LIN {X 0,Y 490.396,Z 454.838,A -85,B 0,C 180,E1 -6677.515,E2 -6677.515} C_VEL
LIN {X 0,Y 490.026,Z 466.047,A -85,B 0,C 180,E1 -6678.176,E2 -6678.176} C_VEL
LIN {X 0,Y 489.6,Z 478.217,A -85,B 0,C 180,E1 -6679.098,E2 -6679.098} C_VEL
LIN {X 0,Y 489.209,Z 488.314,A -85,B 0,C 180,E1 -6680.059,E2 -6680.059} C_VEL
LIN {X 0,Y 488.92,Z 496.882,A -85,B 0,C 180,E1 -6681.061,E2 -6681.061} C_VEL
LIN {X 0,Y 488.59,Z 504.795,A -85,B 0,C 180,E1 -6682.184,E2 -6682.184} C_VEL
LIN {X 0,Y 488.343,Z 512.501,A -85,B 0,C 180,E1 -6683.538,E2 -6683.538} C_VEL
LIN {X 0,Y 488.097,Z 518.492,A -85,B 0,C 180,E1 -6684.888,E2 -6684.888} C_VEL
LIN {X 0,Y 488.028,Z 522.544,A -85,B 0,C 180,E1 -6686.054,E2 -6686.054} C_VEL
LIN {X 0,Y 487.922,Z 526.14,A -85,B 0,C 180,E1 -6687.447,E2 -6687.447} C_VEL
LIN {X 0,Y 487.854,Z 528.078,A -85,B 0,C 180,E1 -6688.505,E2 -6688.505} C_VEL
LIN {X 0,Y 487.819,Z 529.721,A -85,B 0,C 180,E1 -6690.182,E2 -6690.182} C_VEL
LIN {X 0,Y 487.791,Z 529.786,A -85,B 0,C 180,E1 -6691.781,E2 -6691.781} C_VEL
LIN {X 0,Y 487.832,Z 528.402,A -85,B 0,C 180,E1 -6693.322,E2 -6693.322} C_VEL
LIN {X 0,Y 487.904,Z 525.75,A -85,B 0,C 180,E1 -6694.808,E2 -6694.808} C_VEL
LIN {X 0,Y 488.023,Z 521.831,A -85,B 0,C 180,E1 -6696.248,E2 -6696.248} C_VEL
LIN {X 0,Y 488.188,Z 516.599,A -85,B 0,C 180,E1 -6697.646,E2 -6697.646} C_VEL
LIN {X 0,Y 488.364,Z 510.06,A -85,B 0,C 180,E1 -6699.002,E2 -6699.002} C_VEL
LIN {X 0,Y 488.666,Z 501.865,A -85,B 0,C 180,E1 -6700.336,E2 -6700.336} C_VEL
LIN {X 0,Y 489.03,Z 492.334,A -85,B 0,C 180,E1 -6701.574,E2 -6701.574} C_VEL
LIN {X 0,Y 489.386,Z 482.742,A -85,B 0,C 180,E1 -6702.577,E2 -6702.577} C_VEL
LIN {X 0,Y 489.791,Z 471.387,A -85,B 0,C 180,E1 -6703.531,E2 -6703.531} C_VEL
LIN {X 0,Y 490.195,Z 460.329,A -85,B 0,C 180,E1 -6704.268,E2 -6704.268} C_VEL
LIN {X 0,Y 490.613,Z 447.803,A -85,B 0,C 180,E1 -6704.903,E2 -6704.903} C_VEL
LIN {X 0,Y 490.604,Z 437.986,A -85,B 0,C 180,E1 -6705.287,E2 -6705.287} C_VEL
LIN {X 0,Y 488.136,Z 424.452,A -85,B 0,C 180,E1 -6705.746,E2 -6705.746} C_VEL
LIN {X 0,Y 488.2,Z 417.105,A -85,B 0,C 180,E1 -6709.079,E2 -6709.079} C_VEL
LIN {X 0,Y 488.248,Z 410.497,A -85,B 0,C 180,E1 -6712.075,E2 -6712.075} C_VEL
LIN {X 0,Y 487.578,Z 409.095,A -85,B 0,C 180,E1 -6712.745,E2 -6712.745} C_VEL
LIN {X 0,Y 484.743,Z 406.98,A -85,B 0,C 180,E1 -6713.838,E2 -6713.838} C_VEL
LIN {X 0,Y 482.384,Z 405.303,A -85,B 0,C 180,E1 -6714.718,E2 -6714.718} C_VEL
LIN {X 0,Y 481.417,Z 403.914,A -85,B 0,C 180,E1 -6715.396,E2 -6715.396} C_VEL
LIN {X 0,Y 481.362,Z 403.419,A -85,B 0,C 180,E1 -6715.624,E2 -6715.624} C_VEL
LIN {X 0,Y 481.463,Z 396.479,A -85,B 0,C 180,E1 -6718.787,E2 -6718.787} C_VEL
LIN {X 0,Y 481.483,Z 390.136,A -85,B 0,C 180,E1 -6721.679,E2 -6721.679} C_VEL
LIN {X 0,Y 481.659,Z 382.814,A -85,B 0,C 180,E1 -6724.965,E2 -6724.965} C_VEL
LIN {X 0,Y 481.722,Z 380.482,A -85,B 0,C 180,E1 -6726.117,E2 -6726.117} C_VEL
LIN {X 0,Y 481.697,Z 380.482,A -85,B 0,C 180,E1 -6729.501,E2 -6729.501} C_VEL
LIN {X 0,Y 481.69,Z 380.486,A -85,B 0,C 180,E1 -6732.156,E2 -6732.156} C_VEL
LIN {X 0,Y 481.745,Z 380.477,A -85,B 0,C 180,E1 -6734.774,E2 -6734.774} C_VEL
LIN {X 0,Y 481.752,Z 380.479,A -85,B 0,C 180,E1 -6738.214,E2 -6738.214} C_VEL
LIN {X 0,Y 481.762,Z 380.477,A -85,B 0,C 180,E1 -6741.61,E2 -6741.61} C_VEL
LIN {X 0,Y 481.773,Z 380.476,A -85,B 0,C 180,E1 -6744.977,E2 -6744.977} C_VEL
LIN {X 0,Y 481.909,Z 380.458,A -85,B 0,C 180,E1 -6747.491,E2 -6747.491} C_VEL
LIN {X 0,Y 481.952,Z 380.616,A -85,B 0,C 180,E1 -6749.998,E2 -6749.998} C_VEL
LIN {X 0,Y 481.779,Z 385.211,A -85,B 0,C 180,E1 -6752.506,E2 -6752.506} C_VEL
LIN {X 0,Y 481.632,Z 391.452,A -85,B 0,C 180,E1 -6755.861,E2 -6755.861} C_VEL
LIN {X 0,Y 481.465,Z 396.225,A -85,B 0,C 180,E1 -6758.391,E2 -6758.391} C_VEL
LIN {X 0,Y 481.375,Z 403.104,A -85,B 0,C 180,E1 -6761.99,E2 -6761.99} C_VEL
LIN {X 0,Y 481.157,Z 409.754,A -85,B 0,C 180,E1 -6765.416,E2 -6765.416} C_VEL
LIN {X 0,Y 481.026,Z 416.299,A -85,B 0,C 180,E1 -6768.747,E2 -6768.747} C_VEL
LIN {X 0,Y 480.956,Z 421.018,A -85,B 0,C 180,E1 -6771.133,E2 -6771.133} C_VEL
LIN {X 0,Y 482.859,Z 432.162,A -85,B 0,C 180,E1 -6771.56,E2 -6771.56} C_VEL
LIN {X 0,Y 482.889,Z 439.572,A -85,B 0,C 180,E1 -6771.895,E2 -6771.895} C_VEL
LIN {X 0,Y 482.517,Z 451.256,A -85,B 0,C 180,E1 -6772.589,E2 -6772.589} C_VEL
LIN {X 0,Y 482.219,Z 460.784,A -85,B 0,C 180,E1 -6773.339,E2 -6773.339} C_VEL
LIN {X 0,Y 481.904,Z 469.581,A -85,B 0,C 180,E1 -6774.213,E2 -6774.213} C_VEL
LIN {X 0,Y 481.611,Z 477.562,A -85,B 0,C 180,E1 -6775.212,E2 -6775.212} C_VEL
LIN {X 0,Y 481.399,Z 483.94,A -85,B 0,C 180,E1 -6776.205,E2 -6776.205} C_VEL
LIN {X 0,Y 481.112,Z 490.053,A -85,B 0,C 180,E1 -6777.407,E2 -6777.407} C_VEL
LIN {X 0,Y 481.063,Z 495.38,A -85,B 0,C 180,E1 -6778.82,E2 -6778.82} C_VEL
LIN {X 0,Y 480.953,Z 498.039,A -85,B 0,C 180,E1 -6779.788,E2 -6779.788} C_VEL
LIN {X 0,Y 480.825,Z 499.978,A -85,B 0,C 180,E1 -6780.766,E2 -6780.766} C_VEL
LIN {X 0,Y 480.764,Z 501.457,A -85,B 0,C 180,E1 -6782.02,E2 -6782.02} C_VEL
LIN {X 0,Y 480.778,Z 501.75,A -85,B 0,C 180,E1 -6783.569,E2 -6783.569} C_VEL
LIN {X 0,Y 480.848,Z 500.417,A -85,B 0,C 180,E1 -6785.067,E2 -6785.067} C_VEL
LIN {X 0,Y 480.9,Z 499.257,A -85,B 0,C 180,E1 -6785.769,E2 -6785.769} C_VEL
LIN {X 0,Y 481.019,Z 496.866,A -85,B 0,C 180,E1 -6786.798,E2 -6786.798} C_VEL
LIN {X 0,Y 481.089,Z 493.267,A -85,B 0,C 180,E1 -6787.921,E2 -6787.921} C_VEL
LIN {X 0,Y 481.247,Z 489.231,A -85,B 0,C 180,E1 -6788.896,E2 -6788.896} C_VEL
LIN {X 0,Y 481.476,Z 482.706,A -85,B 0,C 180,E1 -6790.13,E2 -6790.13} C_VEL
LIN {X 0,Y 481.748,Z 475.671,A -85,B 0,C 180,E1 -6791.167,E2 -6791.167} C_VEL
LIN {X 0,Y 482.005,Z 467.647,A -85,B 0,C 180,E1 -6792.118,E2 -6792.118} C_VEL
LIN {X 0,Y 482.325,Z 459.037,A -85,B 0,C 180,E1 -6792.933,E2 -6792.933} C_VEL
LIN {X 0,Y 482.701,Z 448.799,A -85,B 0,C 180,E1 -6793.694,E2 -6793.694} C_VEL
LIN {X 0,Y 482.99,Z 437.967,A -85,B 0,C 180,E1 -6794.299,E2 -6794.299} C_VEL
LIN {X 0,Y 482.783,Z 430.957,A -85,B 0,C 180,E1 -6794.61,E2 -6794.61} C_VEL
LIN {X 0,Y 481.007,Z 421.287,A -85,B 0,C 180,E1 -6794.988,E2 -6794.988} C_VEL
LIN {X 0,Y 481.097,Z 415.037,A -85,B 0,C 180,E1 -6798.157,E2 -6798.157} C_VEL
LIN {X 0,Y 481.14,Z 409.349,A -85,B 0,C 180,E1 -6801.09,E2 -6801.09} C_VEL
LIN {X 0,Y 481.265,Z 404.874,A -85,B 0,C 180,E1 -6803.429,E2 -6803.429} C_VEL
LIN {X 0,Y 481.387,Z 399.33,A -85,B 0,C 180,E1 -6806.317,E2 -6806.317} C_VEL
LIN {X 0,Y 481.503,Z 393.756,A -85,B 0,C 180,E1 -6809.279,E2 -6809.279} C_VEL
LIN {X 0,Y 481.657,Z 388.373,A -85,B 0,C 180,E1 -6812.166,E2 -6812.166} C_VEL
LIN {X 0,Y 481.867,Z 383.168,A -85,B 0,C 180,E1 -6814.979,E2 -6814.979} C_VEL
LIN {X 0,Y 481.734,Z 380.484,A -85,B 0,C 180,E1 -6816.598,E2 -6816.598} C_VEL
LIN {X 0,Y 481.674,Z 380.49,A -85,B 0,C 180,E1 -6819.502,E2 -6819.502} C_VEL
LIN {X 0,Y 481.683,Z 380.49,A -85,B 0,C 180,E1 -6822.158,E2 -6822.158} C_VEL
LIN {X 0,Y 481.72,Z 380.484,A -85,B 0,C 180,E1 -6824.775,E2 -6824.775} C_VEL
LIN {X 0,Y 481.776,Z 380.474,A -85,B 0,C 180,E1 -6828.216,E2 -6828.216} C_VEL
LIN {X 0,Y 481.746,Z 380.478,A -85,B 0,C 180,E1 -6831.612,E2 -6831.612} C_VEL
LIN {X 0,Y 481.809,Z 380.471,A -85,B 0,C 180,E1 -6834.14,E2 -6834.14} C_VEL
LIN {X 0,Y 481.913,Z 380.457,A -85,B 0,C 180,E1 -6837.493,E2 -6837.493} C_VEL
LIN {X 0,Y 481.915,Z 380.456,A -85,B 0,C 180,E1 -6840,E2 -6840} C_VEL
LIN {X 0,Y 481.914,Z 380.456,A -85,B 0,C 180,E1 -6842.508,E2 -6842.508} C_VEL
LIN {X 0,Y 481.81,Z 380.472,A -85,B 0,C 180,E1 -6845.861,E2 -6845.861} C_VEL
LIN {X 0,Y 481.741,Z 380.479,A -85,B 0,C 180,E1 -6848.389,E2 -6848.389} C_VEL
LIN {X 0,Y 481.777,Z 380.472,A -85,B 0,C 180,E1 -6851.785,E2 -6851.785} C_VEL
LIN {X 0,Y 481.722,Z 380.481,A -85,B 0,C 180,E1 -6855.225,E2 -6855.225} C_VEL
LIN {X 0,Y 481.695,Z 380.481,A -85,B 0,C 180,E1 -6858.723,E2 -6858.723} C_VEL
LIN {X 0,Y 481.655,Z 380.486,A -85,B 0,C 180,E1 -6861.395,E2 -6861.395} C_VEL
LIN {X 0,Y 481.662,Z 380.486,A -85,B 0,C 180,E1 -6864.114,E2 -6864.114} C_VEL
LIN {X 0,Y 481.731,Z 380.479,A -85,B 0,C 180,E1 -6867.142,E2 -6867.142} C_VEL
LIN {X 0,Y 481.668,Z 380.486,A -85,B 0,C 180,E1 -6869.742,E2 -6869.742} C_VEL
LIN {X 0,Y 481.654,Z 380.489,A -85,B 0,C 180,E1 -6872.676,E2 -6872.676} C_VEL
LIN {X 0,Y 481.625,Z 380.493,A -85,B 0,C 180,E1 -6875.711,E2 -6875.711} C_VEL
LIN {X 0,Y 481.703,Z 380.486,A -85,B 0,C 180,E1 -6879.357,E2 -6879.357} C_VEL
LIN {X 0,Y 481.658,Z 380.491,A -85,B 0,C 180,E1 -6882.16,E2 -6882.16} C_VEL
LIN {X 0,Y 481.646,Z 380.491,A -85,B 0,C 180,E1 -6884.459,E2 -6884.459} C_VEL
